(* CoDeSys 2.3.9.50 project: PLC_1111.pro *)
(* Libraries: standard.lib 5.6.98 12:03:02, TcEtherCAT.lib*1.12.15 17:38:26, TcUtilities.lib 3.2.16 16:08:58, TcBase.lib 14.5.09 12:14:08, FB_DateTime.lib 15.2.16 04:06:26, COMlibV2.lib 24.2.14 00:15:46, TcSystem.lib 7.6.16 11:01:22, TcBaseMath.lib 27.7.04 12:07:56, TcMath.lib 23.9.04 15:15:30, TcSystemCX.lib*6.12.13 20:18:08, SysLibVisu.lib 7.7.04 18:17:22, SysLibTargetVisu.lib 16.6.08 16:24:26, TcSUPS.lib 7.6.16 11:50:06 *)

(* Global variable list: Alarms *)
VAR_GLOBAL

	bFeedinfCylFwdRsError:BOOL;
	bErrorRstHmi:BOOL;

	bAGripperConeAllignError: BOOL;
	bAGripCheckDownBuzzer: BOOL;
	sMessage_ServoGripperDown: STRING;

	bQACartonFeedingPistonValve1: BOOL;
	bQACartonFeedingPistonValve2: BOOL;
	bQACartonStopPiston: BOOL;

	bA3COneCrossed: BOOL;
	bA6ConeCrossed: BOOL;
	c18_ConeCounter1: CTU;
	bMCCycleStarted: BOOL;
	bAError: BOOL;
	bAError1: BOOL;
	bSeparatorVerticalPistonEndRsSensed: BOOL;
	bChkEndSensor: BOOL;
	bAConeFeddCylFwdRsError: BOOL;
	bAWrap_1PistRsError: BOOL;
	bAWrap_2PistRsError: BOOL;
	bAWrap_3PistRsError: BOOL;
	bAForwPistRsError: BOOL;
	bASealTopRsError: BOOL;
	bASealTopPistRsError: BOOL;
	bASealSepaX_axisRsError: BOOL;
	bASealSepaY_axisRsError: BOOL;
	bATiltPistRsError: BOOL;
	bAReversPistnRsError: BOOL;
	bAColumnPushPistnRsError: BOOL;
	bAConeEjectPistnRsError: BOOL;
	bASepaHoriForwdFwdEndRsError: BOOL;
	bASepaHoriForwdEndRsError: BOOL;
	bASepaVertiEndPistnRsError: BOOL;
	bASepaHoriRevValveRsError: BOOL;
	bALenghtTightHomeSenRsError: BOOL;
	bABreadthTightHomeSenRsError: BOOL;
	bAGrossWtSenRsError: BOOL;
	bACartonSenRsError: BOOL;
	HmiEmptyCartonPiston: STRING(80);
	bAWrap_PistRsError: BOOL;
	bASealBottomRsError: BOOL;
	SealTopBottomRsError: BOOL;
	SealConeMiss: STRING;
	bConeMissBit: BOOL;
	bAColoumnConeSenError: BOOL;
	bASepVerticalCylRevRsErrChkBit: BOOL;
	bASepaVerCylhomeRsError: BOOL;
	bAL_BTightHomeSenRsError: BOOL;
	GrossWtReedSwBit: BOOL;
	bAGrossWtHomeSenRsError: BOOL;
	bARowStoppHomeSenRsError: BOOL;
	bAPolythinSheetError: BOOL;
	bASepVerticalCylEndRsErrChkBit: BOOL;
	bASupplyPressureError: BOOL;
	baConePtrsentAtWrapConv: BOOL;
	bSealConveyerConePresent: BOOL;
	HmiConeAtSealConveyer: STRING;
	bConeAtMatrixConveter: BOOL;
	bCartonFullDetectbit: BOOL;
	SeparatorAlertbit: BOOL;
	bAFlimNotLoaded: BOOL;
	bFilmErrClear: BOOL;
	bAFirst3ConeAtRowConeCount: BOOL;
	bGrossWieghtNokTemp: BOOL;
	GrossWtAlarm: STRING;
	SealingUnitAlert: BOOL;
	PressureSeparatorAlert: BOOL;
	PistonAlertAlarm: BOOL;
	GripperUnitAlert: BOOL;
	GrossWeightAlert: BOOL;
	ERROR_ALERT: BOOL;
	SealBitAlert: BOOL;
	bAConeMissAtMatricConv: BOOL;
	bHmiColourChangeBit: BOOL;
	bHmiColourChangeBit2: BOOL;
	bAConeAtFullConveyor: BOOL;
	bEmptyCartonDetectError: BOOL;
	HMIEmptyCartonDetectErr: STRING;
	bAEmergencyPressed: BOOL;
	bAConeMissErrorAtWrpConv: BOOL;
	bWrapConvStopped2: BOOL;
	bACheckWrappConvError1: BOOL;
	bACheckWrappConvError2: BOOL;
	bACheckWrappConvError3: BOOL;
	bACheckWrappConvError4: BOOL;
	InterLockCounterRESET: BOOL;
	bCone1LockBit: BOOL;
	bA6conesPushedTemp: BOOL;
	bAConeFeedCylStart: BOOL;
	bWrapConvStopped3: BOOL;
	bAByPassOn2: BOOL;
	bConeMiss3AtWrapConv: BOOL;
	bWrapConvStopped4: BOOL;
	bConeMiss4AtWrapConv: BOOL;
	bAWrapConeCyl123_23: BOOL;
	bCount_ConvLockBit: BOOL;
	bCount_ConvLockBit2: BOOL;
	bCount_ConvLockBitTemp: BOOL;
	FileCreateTemp: BOOL;
	rGrossWeighToReport: REAL;
	bServoOff: BOOL;
	sSupplyPressuremsg: STRING;
	bTLBlinkOn: BOOL;
	PopUp: BOOL;
	bAByPassOn3: BOOL;
	bConeMiss2AtWrapConvtEMP: BOOL;
	CountB_Hmi: INT;
	bA3ConeCrossed_24: BOOL;
	SealBitAlert_24: BOOL;
	bAFilm1Loaded_24_7Cone: BOOL;
	bAFilm1Loaded_24_6Cone: BOOL;
	bAFilm1Loaded_24_5Cone: BOOL;
	bAFilm1Loaded_24_4Cone: BOOL;
	bAFilm1Loaded: BOOL;
	bAFilm2Loaded: BOOL;
	bAFilm3Loaded: BOOL;
	bAFilm1Loaded_24_8Cone: BOOL;
	SealingSafety: BOOL;
	bACheckWrappConvError5: BOOL;
	SensorCheck123: BOOL;
	bAConeMissErrorAtWrpConvTemp1_24: BOOL;
	bAConeMissErrorAtWrpConvTemp2_24: BOOL;
	bAConeMissErrorAtWrpConvTemp3_24: BOOL;
	bAConeMissErrorAtWrpConvTemp4_24: BOOL;
	SensorCheck56: BOOL;
	SensorCheck78: BOOL;
	bWrapConvStopped3_24: BOOL;
	bWrapConvStopped4_24: BOOL;
	bAConeMissErrorAtWrpConvTemp5_24: BOOL;
	bWrapConvStopped4_24exp: BOOL;
	bWrapConvStopped1_24exp: BOOL;
	TON_4_24: TON;
	TON_6_24: TON;
	TON_8_24: TON;
	TON_5_24: TON;
	TON_9_24: TON;
	TON_10_24: TON;
	TON_11_24: TON;
	TON_12_24: TON;
	TON_13_24: TON;
	mybit2: BOOL;
	HmiFullCartonAtConveyer_sensor: STRING;
	bHmiColourChangeBit2_24: BOOL;
	AlarmBitArray: STRING;
	bACheckWrappConv: BOOL;
	var_7: STRING;
	bAinterlockinit: BOOL;
	bAConvStartBit: BOOL;
	test50: BOOL;
	bANo_ErrorBit: BOOL;
END_VAR

(* Global variable list: Common *)
VAR_GLOBAL

	bConeAtWrppingConveyor: BOOL;
	sendOver1:BOOL;
	sendOver2:BOOL;
	sendOver3:BOOL;
	sendOver4:BOOL;
	b2_4SetHmi: BOOL;
	tSealDyl: TIME;
	SealDelay: TON;
	b3ConeSealOver: BOOL;
	bIConeCountSensorVal: INT;
	SealDelay1: TON;
	tSealDyl1: TIME;
	SealDelay2: TON;
	tSealDyl2: TIME;
(*============El6022=================*)

	sSendString : STRING;
	sRecvString : STRING;
	nSendASC:BYTE;
	(* 	I/O variables for a PC-COM port *)

	bAConeUnderWeight: BOOL;
	iACounterA_PV: INT;
	bACounterAReset: BOOL;
	bACounterBReset: BOOL;
	iACounterB_PV: INT;
	iACounterTilt_PV: INT;
	bAresetHmi: BOOL;
	CounterTilt: CTU;
	bAtiltGoHome: BOOL;
	bA5thConeFeedStart: BOOL;
	bAWrappingConvStartAuto: BOOL;
	bAWrappingConvStart: BOOL;
	bAWrappingConvStart1: BOOL;
	bAWrappingConvStart2: BOOL;
	bAWrappingConvStart3: BOOL;
	bAWrappingConvStart4: BOOL;
	bAWrappingConvStart5: BOOL;
	bAWrapConeCyl2: BOOL;
	bA3ConeWrappOver: BOOL;
	bASeal3ConeStart: BOOL;
	bA8thConeWrappOver: BOOL;
	bA6thConeWrappOver: BOOL;
	bA4thWrappOver: BOOL;
	bAutoModeHmi: BOOL;
	bManualModeHmi: BOOL;
	bAColumnPushPistonStart1: BOOL;
	bAColumnPushPistonStart2: BOOL;
	bAMatrixConvStart1: BOOL;
	bAMatrixConvStart2: BOOL;
	bARowStopperMotorRevStart: BOOL;
	bAGripperSeqover: BOOL;
	bAServoDownDone: BOOL;
	bAServoDownDone2: BOOL;

(*

	iarrEcMasterNetId AT %I*: T_AmsNetIdArr;
	nEcMasterSlaveCountCfg AT %I*: UINT;
	bStart: BOOL;
	nTotalSlaves: INT;
	nSalveinfo: ARRAY [0..ISLAVEADDR_ARR_SIZE] OF ST_SlaveStateInfo;
	Iout1 AT%Q*:BOOL;
*)
(*test======*)


	FB_EcGetAllSlaveStates: FB_EcGetAllSlaveStates;
	bEthrcatinfo: BOOL;
	All_slave_Staus_Busy: BOOL;
	All_slave_Staus_Err: BOOL;
	All_slave_Staus_Err_ID: UDINT;
	iNumOfSlavesRead: INT;
	arrSlaveStates: ARRAY [0..10] OF ST_EcSlaveState;

	bAEmptyCartonConvContinue: BOOL;
	bA4thConeFeedStart23: BOOL;
	bA4thConeFeedStartAuto23: BOOL;
	bA6thConeFeedStartAuto23: BOOL;
	bAtiltGoHome3_23: BOOL;

	CounterTilt23: CTU;
	bAtiltGoHome2_23: BOOL;
	bAtiltGoHome1_23: BOOL;
	bAWrappingConvStart1_23: BOOL;
	bAWrappingConvStart4_23: BOOL;
	bAWrappingConvStart3_23: BOOL;
	bAWrappingConvStart2_23: BOOL;
	bA6ConeWrappOver23: BOOL;
	bAColumnPushPistonStart2_23: BOOL;
	bAColumnPushPistonStart1_23: BOOL;

	bAConvFirstStart: BOOL;
	bAServoFwdStart: BOOL;
	bAServoUpAuto: BOOL;
	bAConePickDone: BOOL;
	bAServoDown1Done: BOOL;

	bAPlaceOver: BOOL;
	bAServoFwdStart2: BOOL;
	bAConvSecStart: BOOL;
	bAUnitAWeighOk: BOOL;
	bASeparatorUnitEnable: BOOL;
	bAServoUpDone: BOOL;

	bAFirstSetToMatrix: BOOL;
	bAConvFirstStartUnitB: BOOL;
	bAUnitBWeighOk: BOOL;

	bAConvSecStartUnitB: BOOL;
	bQAFeedingConveyorMotorB: BOOL;
	bQAFeedingConveyorMotorA: BOOL;
	bA3Pushed: BOOL;
	bAconvReayTemp: BOOL;
	bAconvReayTemp2: BOOL;
	bA6conesPushed: BOOL;
	WCPReady: BOOL;
	InterLockCounter: CTU;
	bATiltEnable1: BOOL;

	InterLockCounterStart: BOOL;
	bAWrapConvStarted: BOOL;
	bAInterlockCountStart: BOOL;


	b4thConePushed: BOOL;
	bAconvReayTemp3: BOOL;
	bAconvReadyTemp3: BOOL;
	b6thConePushed_24: BOOL;
	bAconvReadyTemp4: BOOL;
	b8thConesPushed: BOOL;
	bAconvReadyTemp5: BOOL;
	bATiltEnable1_24: BOOL;
	bAConeFeedPistonLockOk: BOOL;

	bATiltEnable2_24: BOOL;
	bAWrapConvReady_24: BOOL;
	bATiltEnable3_24: BOOL;
	bACartonReady_24: BOOL;
	bAResetEnabled: BOOL;
	bRFwdRevPistonRst: BOOL;
	bRTiltPistonReset: BOOL;
	CounterTilt23Rst1: BOOL;
	bACartonReady_23: BOOL;
	bResetRowStopper: BOOL;

	bSealConvIntOver: BOOL;
	bSealConvStart: BOOL;
	bSealConvStart1: BOOL;
	bSealConvStart2: BOOL;
	bASecondSetToMatrix: BOOL;
	bSealConvStart3: BOOL;
	bAConvReady: BOOL;
	bASealConvEnd1: BOOL;
	bASealConvEnd2: BOOL;
	bSaelUnitIntOver: BOOL;
	bWCSStart1: BOOL;
	bWCSStart2: BOOL;
	bWCSStart3: BOOL;
	bMCStart1: BOOL;
	bOneSetReached: BOOL;
	bMCStart2: BOOL;
	bRowStopperAt23Pos: BOOL;
	bATiltPistonInHome: BOOL;
	bSealConvStart1_24: BOOL;
	bSealConvStart2_24: BOOL;
	bSealConvStart3_24: BOOL;
	bASealConvEnd1_24: BOOL;
	bASealConvEnd2_24: BOOL;
	bWCSStart1_24: BOOL;
	bWCSStart2_24: BOOL;
	bRowStopperAt24Pos: BOOL;
	iarrEcMasterNetId: T_AmsNetIdArr ;
	nEcMasterSlaveCountCfg AT %I*: UINT;
	nSalveinfo: ARRAY [0..ISLAVEADDR_ARR_SIZE] OF ST_SlaveStateInfo;

	iRemote2State: INT;
	bRetUnitAStart: BOOL;
	bUnitARowStopperStarted: BOOL;
	bMCStartInAuto: BOOL;
	bStartCartonCov: BOOL;
	bAStartCartonCov: BOOL;

	bRetUnitBStart: BOOL;
	bUnitBRowStopperStarted: BOOL;
	bAOneMinConvStart: BOOL;
	bStartConeFeedConvInBypass: BOOL;
	bUnitBCounterRst: BOOL;
	bASeparatorUnitEnable3: BOOL;
	bASeparatorUnitEnable2: BOOL;
	bASeparatorUnitEnable1: BOOL;
	bQARowStopperMotorRev1: BOOL;
		bAConeOnMatrixConv: BOOL;
	HmiConeOnMatxConvey: STRING;
	bAFilmLoadedCom: BOOL;
	HmiPolyThinFeedErr: STRING;
	bARCartanConvOn: BOOL;
	bOneMinConvOver: BOOL;
	bAWrapConeCyl123: BOOL;
	bAByPassOn: BOOL;
	bA6thConeFeedStart23: BOOL;
	iTotalLayers: INT;
	Count_Hmi: DINT;
	SealingOver: BOOL;
	SealingOver1: BOOL;
	bAFirstConeReached: BOOL;
	Interlockfor_1Cone_24: BOOL;
	Interlockfor_5Cone_24: BOOL;
	Interlockfor_7Cone_24: BOOL;
	UnitACone3Sensing: BOOL;
	UnitACone2Sensing: BOOL;
	UnitACone1Sensing: BOOL;
	UnitACone1_Move: BOOL;
	UnitACone1Sensing_2: BOOL;
	UnitACone2Sensing_2: BOOL;
	UnitACone3Sensing_2: BOOL;
	UnitACone2_Move: BOOL;
	UnitACone3_Move: BOOL;
	UnitA_3_ConeSensed: BOOL;
	R_TRIG_3ConeSensing: R_TRIG;
	iATotalNoOfCones: INT;
	bAUnitBConeCrossing_24: BOOL;
	UnitAConeCrossCount: CTU;
	UnitBCompleteCheckCount_24: CTU;
	Message1_24: STRING;
	sMessage_24: STRING;
	sMessage_23: STRING;
	sMessage_23_Feeding: STRING;
	sMessage_23_Forwad_rev: STRING;
	sMessage_23_Tilting: STRING;
	sMessage_Wrapping: STRING;
	sMessage_Sealing: STRING;
	sMessage_Colomn: STRING;
	sMessage_Gripper: STRING;
	sMessage_Carton: STRING;
	sMessage_Separator: STRING;
	(*FB_S_UPS_CX51x0_1: FB_S_UPS_CX51x0;*)
	bACheckWrappConvError1_23: BOOL;
	bACheckWrappConvError4_23: BOOL;
	bACheckWrappConvError2_23: BOOL;
	bACheckWrappConvError3_23: BOOL;
	mybit1: BOOL;
	temp1: REAL;
	temp2: REAL;
	temp3: REAL;
	temp4: REAL;
	mybit3: BOOL;
	mybit4: BOOL;
	var_1: REAL;
	var_5: REAL;
	bAFeedingConvOff: BOOL;
	bAFeedingConvOff_1: BOOL;
	bQSealBitAlert: BOOL;
	bQSealBitAlert_24: BOOL;
	bA3ConeWrappOver_24: BOOL;
	SealConeMissAlet_24: BOOL;
END_VAR


VAR_GLOBAL CONSTANT
	iSLAVEADDR_ARR_SIZE:DINT:= 256;
END_VAR
(*
VAR_GLOBAL RETAIN
	iTotalLayersHold AT %Q*: INT;
END_VAR *) 
VAR_GLOBAL PERSISTENT
	iTotalLayersHold: INT;
END_VAR

(* Global variable list: Hmi *)
VAR_GLOBAL
	bAllOuputOff: BOOL;
(*	sSettingArray AT %Q*:ARRAY[0..20] OF SETTING; *)
	i:INT;
	sMillNameHmi: STRING(80) := 'INDO TEXNOLOGY';
	AddressLine1Hmi: STRING(80);
	AddressLine2Hmi: STRING(80);
	AddressLine3Hmi: STRING;
	sAddressLine1Hmi: STRING(80) :=' ONDIPUDUR';
	sAddressLine2Hmi: STRING(80) := 'COIMBATORE';
	sAddressLine3Hmi: STRING(80) := 'INDIA';
	bEmptyConeSubOnHmi: BOOL;
	bEmptyConeSubEnabled: BOOL;
	bEmptyConeSubOffHmi: BOOL;
	bAutoRetrivalOnHmi: BOOL;
	bAutoRetrivalEnabled: BOOL;
	bAutoRetrivalOffHmi: BOOL;
	bPrintAutoOnHmi: BOOL;
	bPrintAutoEnabled: BOOL;
	bPrintAutoOffHmi: BOOL;
	PrintDefaultWeightOnHmi: BOOL;
	PrintDefaultWeightOnEnabled: BOOL;
	PrintDefaultWeightOffHmi: BOOL;
	NegToleranceOnHmi: BOOL;
	NegToleranceEnabled: BOOL;
	NegToleranceOffHmi: BOOL;



	Recipe_Var: ARRAY [1..2] OF Recipe;

	DateTimeVar: STRING;
	LogMonth: STRING(80);
	LogYear: STRING(80);
	logDay: STRING(80);
	sStation1ActiveAlarms: STRING(80);
	OperatorName: STRING;

	bEmptyConeSubEnableHMI: BOOL;
	bAEmptyConeSubEnabled: BOOL;
	bEmptyConeSubDisableHMI: BOOL;
	bAutoRetrivalEnableHMI: BOOL;
	bAAutoRetrivalEnabled: BOOL;
	bAutoRetrivalDisableHMI: BOOL;
	bAutoPrintEnableHMI: BOOL;
	bAAutoPrintEnabled: BOOL;
	bAutoPrintDisableHMI: BOOL;
	bDefaultWeighPrintEnableHMI: BOOL;
	bDefaultWeighPrintDisableHMI: BOOL;
	bADefaultWeighPrintEnabled: BOOL;
	bNegToletanceEnableHMI: BOOL;
	bNegToletanceDisableHMI: BOOL;
	bANegToletanceEnabled: BOOL;
	bADayComplete: BOOL;
	bADayStart: BOOL;
	bAutoSealingEnableHMI: BOOL;
	bAAutoSealEnabled: BOOL;
	sCityTownHmi: STRING(80);
	sCountryHmi: STRING(80);
	GrossWeightHmi: REAL;
	NetToleranceHmi: REAL;
	sDescriptionHmi: STRING(80);
(*	SCountHmi: INT;  *)

	iCountHmi: STRING;
	iCartoNoHmi: INT;
	sPackingTypeHmiTemp: STRING(80);
	sMaterialTypeHmiTemp: STRING(80);
	iConeDiaHmi: INT;
	iHieghtHmi: INT;
	iWeightHmi: INT;
	iTipColorHmi: STRING;
	INoOfRowsHmi: INT;
	iNoOfColoumsHmi: INT;
	NoOfLayersHmi: INT;
	iCortonWeightHmi: INT;
	iCartonHmi: INT;
	iLenghtHmi: INT;
	iNoOfConeHmi: INT;
	iNetWeightHmi: REAL;


(*==================*)


	bBlink_Time: BOOL;
	File_Path: STRING;

	bCloseAttachmentList: BOOL;
	bPauseHmi: BOOL;
	bAPauseSeq: BOOL;
	bResumeHmi: BOOL;


	sStringArray:ARRAY [1..cnMaxStrings] OF STRING(300);

	Pgm_NoHmi: INT;
	bNoHmi: BOOL;
	bHidePopUp: BOOL;
	bPauseYesHmi: BOOL;
	bPauseNoHmi: BOOL;

	SealComDlyTemp: TIME;
	wTodayToHmi: STRING;
	bLoadPgm: BOOL;
	bLoadPgmHmi: BOOL;
	bAutoSealingHmi: BOOL;
	bAutoSealOn: BOOL;
	bCartonPackingOn: BOOL;
	bPallettePackingOn: BOOL;
	bCartonPackingHmi: BOOL;
	bPallettePackingHmi: BOOL;
	bConeHmi: BOOL;
	bConeOn: BOOL;
	bCheeseOn: BOOL;
	bCheeseHmi: BOOL;
	bNewRecipeHmi: BOOL;
	Var_PgmNo: INT;
	Var_Description: STRING;

(*==========new variables===========*)
	SaveRecipeHmi: BOOL;
	bCreateNew: BOOL;
	PgmNoDis1: INT;
	PgmNameDis: STRING;
	bModel1Hmi: BOOL;
	PgmNameDis1: STRING(80);
	PgmNameDis2: STRING(80);
	bModel2Hmi: BOOL;
	PgmNoDis3: INT;
	PgmNameDis3: STRING;
	PgmNoDis4: INT;
	PgmNameDis4: STRING;
	PgmNoDis5: INT;
	PgmNoDis6: INT;
	PgmNameDis5: STRING;
	PgmNameDis6: STRING;
	bModel3Hmi: BOOL;
	bModel4Hmi: BOOL;
	bModel5Hmi: BOOL;
	bModel6Hmi: BOOL;
	bEditRecipeHmi: BOOL;
	bEditRecipeEnabled: BOOL;
	bSaveRecipeHmi: BOOL;
	rPickPosMinHmi: REAL := 0.00;
	iDropVeloHmi: REAL;
	PosAct: DINT;
	rServiActPosHmi: REAL;
	b2_3SetHmi: BOOL;
	diVeloActHmi: DINT;
	bStopHmi: BOOL;
	bRetUnitARst: BOOL;
	bGripperOpenHmi: BOOL;
	bGrippercCloseHmi: BOOL;
	sMCStatus: STRING;
	iDropPosHmi: REAL;
	bJogNegHmi: BOOL;
	bJogPositiveHmi: BOOL;
	bJogNegativeHmi: BOOL;
	sRetreivalAStatus: STRING;
	sRetreivalBStatus: STRING;
	bGWPistonOnHmi: BOOL;
	bGWPistonOffHmi: BOOL;
	bRCOnHmi: BOOL;
	bRCOffHmi: BOOL;
	bWeightAckHmi: BOOL;
	bInitializeHmi: BOOL;
	bServoHomeHmi: BOOL;
	rGrossWtTolHmi: REAL;
	bRstHmi: BOOL;
	OpCountHmi: INT;
	bloadRecipeHmi: BOOL;
	rGrossTollHmi: REAL;
	iAPartCountToHmi AT %Q*: INT;
	HmiYAxisPiston: STRING(80);
	HmiXAxisPiston: STRING(80);
	HMISealTopPiston: STRING(80);
	HMISealBotPiston: STRING(80);
	HMIForwdPiston: STRING(80);
	HMIFeedPiston: STRING(80);
	HMIWrapPiston1: STRING(80);
	HMIWrapPiston2: STRING(80);
	HMIWrapPiston3: STRING(80);
	ConeMissAlarm: STRING(80);
	bErrorReset: BOOL;
	HmiTiltPiston: STRING(80);
	HmiReverPiston: STRING(80);
	HmiColuPushrPiston: STRING(80);
	HmiConeEjePiston: STRING(80);
	HmiSepHorizPiston: STRING(80);
	HmiSepVertiPiston: STRING(80);
	HmiSepHoriRevPiston: STRING(80);
	HmiLengthPiston: STRING(80);
	HmiBreadthPiston: STRING(80);
	HmiServoHome: STRING(80);
	HmiGrossWtPiston: STRING(80);
	HmiColoumConeSen: STRING;
	HmiSepVeticCylHomeRsError: STRING;
	HmiGrossWtHomePiston: STRING;
	HmiWrapConvStatus: STRING;
	HmiConeAtMatrixConveyer: STRING;
	HmiFullCartonAtConveyer: STRING;
	bAIntStarted: BOOL;
	HMISeparatorPaperDetec: STRING;
	CounterTilt23_CV_HMI: INT;
	HmiFilmLoadErr: STRING;
	bSheetNotFeeded: STRING;
	bEmergency: BOOL;
	sDATEFinal: STRING;
	sShitToReport: STRING;
	sFinalGrossWt: STRING(80);
	bAIntBlinkAuto: BOOL;
	bALayer1Selected: BOOL;
	bALayer2Selected: BOOL;
	bALayer3Selected: BOOL;
	bMCCycleStartedHold: BOOL;
	RowStopperCountvalue: DINT;



	iLotNoHmi: DWORD;
	bStopEnable: BOOL;
	ITotalSample: DINT;
	iCartonSample: DWORD;
END_VAR
VAR_GLOBAL CONSTANT
	MAX_CSV_ROWS 			: UDINT := 100;
	MAX_CSV_COLUMNS 		: UDINT := 5;
	MAX_CSV_FIELD_LENGTH	: UDINT := 100;

	cnMaxStrings:	INT:=1000;




END_VAR
(*
VAR_GLOBAL RETAIN
	iPickPosHmi AT %Q*: REAL;
	rPickVeloHmi AT %Q*: REAL;
	rDropVeloHmi AT %Q*: REAL;
	iDropPos1Hmi AT %Q*: REAL;
	iDropPos2Hmi AT %Q*: REAL;
	iDropPos3Hmi AT %Q*: REAL;


	bLayer1SelectHmi AT %Q*: BOOL;
	bLayer2SelectHmi AT %Q*: BOOL;
	bLayer3SelectHmi AT %Q*: BOOL;
	iTotalCones AT %Q*: DINT;
END_VAR*)
VAR_GLOBAL PERSISTENT
	iTotalCones: DINT;
	iPickPosHmi: REAL;
	rPickVeloHmi: REAL;
	rDropVeloHmi: REAL;
	iDropPos1Hmi: REAL;
	iDropPos2Hmi: REAL;
	iDropPos3Hmi: REAL;
	bLayer1SelectHmi: BOOL;
	bLayer2SelectHmi: BOOL;
	bLayer3SelectHmi: BOOL;
	sSettingArray: ARRAY [0..20] OF SETTING;
	bAShift1Hour: BOOL;
	bAShift2Hour: BOOL;
	bAShift3Hour: BOOL;
	Shift1MinFrom_HMI: WORD;
	Shift2MinFrom_HMI: WORD;
	Shift3MinFrom_HMI: WORD;
	Shift1MinTo_HMI: WORD;
	Shift2MinTo_HMI: WORD;
	Shift3MinTo_HMI: WORD;
	Sfiht1From_Hmi: WORD;
	Sfiht2From_Hmi: WORD;
	Sfiht3From_Hmi: WORD;
	Sfiht1To_Hmi: WORD;
	Sfiht2To_Hmi: WORD;
	Sfiht3To_Hmi: WORD;
END_VAR

(* Global variable list: Inputs_Gripper *)
VAR_GLOBAL



(******************EL1809(Gripper)*********************)



	bIColumnconeDetection AT %I*: BOOL;
	bIColumnPushPistonHome AT %I*: BOOL;
	bIColumnPushPistonEnd AT %I*: BOOL;
	bIRowConeCountSensor AT %I*: BOOL;
	bIRowConeDetection AT %I*: BOOL;
	bIColumnStopperHome AT %I*: BOOL;
	bIColumnStopper1 AT %I*: BOOL;
	bIColumnStopper2 AT %I*: BOOL;

	bIColumnStopper3 AT %I*: BOOL;
	bIRowStopperHome AT %I*: BOOL;
	bIRowStopper1 AT %I*: BOOL;
	bIRowStopper2 AT %I*: BOOL;
	bIRowStopper3 AT %I*: BOOL;
	bICartonFeedingPistonHome AT %I*: BOOL;
	bICartonFeedingPistonEnd AT %I*: BOOL;
	bIEmptyCartonDetectionSensor AT %I*: BOOL;




(******************EL1809(Gripper)*********************)




	bISeparatorDetectionSensor AT %I*: BOOL;
	bISeparatorPickupDetectionSensor AT %I*: BOOL;
	bICartonPosition1 AT %I*: BOOL;
	bICartonPosition2 AT %I*: BOOL;
	bICartonPosition3 AT %I*: BOOL;
	bISeparatorHorizontalPistonHome AT %I*: BOOL;
	bISeparatorHorizontalPistonEnd AT %I*: BOOL;
	bISeparatorVerticalPistonHome AT %I*: BOOL;


	bISeparatorVerticalPistonEnd AT %I*: BOOL;
	bIGripperVerticalHome AT %I*: BOOL;
	bIGripperVerticalEnd AT %I*: BOOL;
	bILengthTightPistonHome AT %I*: BOOL;
	bIBreadthTightPistonHome AT %I*: BOOL;
	bIConeEjectionPistonHome AT %I*: BOOL;
	bIConeEjectionPistonEnd AT %I*: BOOL;
	bIFullCartonCountingSensor AT %I*: BOOL;


(******************EL1004(Gripper)*********************)

	bIGrossWtDeductSensor AT %I*: BOOL;
	bIGrossWtPistonHome AT %I*: BOOL;
	bIGrossWtPistonEnd AT %I*: BOOL;
	bIGripperConeDetection AT %I*: BOOL;

	iActCounter AT %I*: UDINT;


	b2_3_ACaron: BOOL;
	b2_3_BCarton: BOOL;
	b2_3_ACarton: BOOL;

END_VAR

VAR_GLOBAL PERSISTENT
	b2_3_ACartonHMI: BOOL;
	b2_3_BCartonHMI: BOOL;
END_VAR

(* Global variable list: Inputs_Main *)
VAR_GLOBAL


(******************EL1809(Matrix)*********************)

	bIConeFeedingPistonHome AT %IX0.0: BOOL;
	bIConeFeedingPistonEnd AT %IX0.1: BOOL;
	bIConeOrientationTop AT %IX0.2: BOOL;

	bIForwardPistonHome AT %IX0.3: BOOL;
	bIForwardPistonEnd AT %IX0.4: BOOL;
	bIReversePistonHome AT %IX0.5: BOOL;
	bIReversePistonEnd AT %IX0.6: BOOL;
	bITiltingHome AT %IX0.7: BOOL;
	bITiltingEnd AT %IX1.0: BOOL;
	bIWrappingChannelPiston1_Home AT %IX1.1: BOOL;
	bIWrappingChannelPiston1_End AT %IX1.2: BOOL;
	bIWrappingChannelPiston2_Home AT %IX1.3: BOOL;
	bIWrappingChannelPiston2_End AT %IX1.4: BOOL;
	bIWrappingChannelPiston3_Home AT %IX1.5: BOOL;
	bIWrappingChannelPiston3_End AT %IX1.6: BOOL;
	bISpare AT %IX1.7:BOOL;

(******************EL1809(Matrix)*********************)

	bIWrappingCone1 AT %IX2.0: BOOL;
	bIWrappingCone2 AT %IX2.1: BOOL;
	bIWrappingCone3 AT %IX2.2: BOOL;
	bIWrappingFilmTensionPlate_1 AT %IX2.3: BOOL;
	bIWrappingFilmTensionPlate_2 AT %IX2.4: BOOL;
	bIWrappingFilmTensionPlate_3 AT %IX2.5: BOOL;
	bISealingTopPistonHome AT %IX2.6: BOOL;
	bISealingTopPistonEnd AT %IX2.7: BOOL;
	bISealingBottomPistonHome AT %IX3.0: BOOL;
	bISealingBottomPistonEnd AT %IX3.1: BOOL;
	bIConeCountSensor AT %IX3.2: BOOL;
	bISealingSeparatorYAxisHome AT %IX3.3: BOOL;
	bISealingSeparatorYAxisEnd AT %IX3.4: BOOL;
	bISealingSeparatorXAxisHome AT %IX3.5: BOOL;
	bISealingSeparatorXAxisEnd AT %IX3.6: BOOL;
	bIManualSealing  AT %IX3.7: BOOL;

(******************EL1809(Matrix)*********************)

	bISealingReverseConeSwitch  AT %IX4.0: BOOL;
	bIPressureSwitch   AT %IX4.1: BOOL;
	bIEmergencySwitch   AT %IX4.2: BOOL;
	bIKeySwitch AT %IX4.3: BOOL;
	bIAutoManual AT %IX4.4: BOOL;
	bIMcStart AT %IX4.5: BOOL;
	bIMcStop AT %IX4.6: BOOL;

(**************************End***********************************)



	statusWord AT %I*: UINT;
	bConeMiss1AtWrapConv: BOOL;
	bConeMiss2AtWrapConv: BOOL;
END_VAR

(*
VAR_GLOBAL PERSISTENT
	SealComDly1 AT %Q*: INT;
END_VAR
VAR_GLOBAL RETAIN PERSISTENT
	ghjnk AT %Q*: INT;
END_VAR
*)



VAR_GLOBAL PERSISTENT
	SealComDly1: INT;
	ghjnk: INT;
END_VAR

(* Global variable list: Inputs_RetrivalA_B *)
VAR_GLOBAL

(*******************EL1809(Retrival A & B )*********************)

	bIUnitA_RowStopperHome  AT %IX10.0: BOOL;
	bIUnitA_RowStopperEnd	 AT %IX10.1: BOOL;
	bIUnitB_RowStopperHome	 AT %IX10.2: BOOL;
	bIUnitB_RowStopperEnd	 AT %IX10.3: BOOL;
	bIUnitA_StartPB 		AT %IX10.4: BOOL;
	bIUnitB_StartPB  		AT %IX10.5: BOOL;
	bIUnitB_LiftPistonHome		AT %IX10.6: BOOL;
	bIUnitB_LiftPistonEnd 		AT %IX10.7:BOOL;
	bIUnitAConedetection1 		AT %IX11.0: BOOL;
	bIUnitAConedetection2		 AT %IX11.1: BOOL;
	bIUnitAConedetection3 AT %IX11.2: BOOL;
	bIUnitAConeCrossing AT %IX11.3: BOOL;
	bIUnitBConedetection1  AT %IX11.4: BOOL;
	bIUnitBConedetection2  AT %IX11.5: BOOL;
	bIUnitBConedetection3 AT %IX11.6: BOOL;
	bIUnitBConeCrossing AT %IX11.7:BOOL;

(******************EL1004(Retrival A & B )*********************)

	bIUnitC_LiftPistonHome AT %IX12.0:BOOL;
	bIUnitC_LiftPistonEnd  AT %IX12.1:BOOL;
	bIUnitC_CartonStopForWeight AT %IX12.2:BOOL;
	bISapre14 AT %IX12.3:BOOL;
END_VAR

(* Global variable list: Manual *)
VAR_GLOBAL




		bQMConeFeedingPistonValve :BOOL;
		bQMForwardPistonValve  :BOOL;
		bQMReversePistonValve :BOOL;
		bQMWrappingChannelPistonValve1:BOOL;
		bQMWrappingChannelPistonValve2:BOOL;
		bQMWrappingChannelPistonValve3 :BOOL;
		bQMSealingTopPistonValve :BOOL;
		bQMSealingBottomPistonValve:BOOL;


		bQMFeedingConveyorMotor :BOOL;
		bQMWrappingConveyorMotor :BOOL;
		bQMSealingConveyorMotor :BOOL;
		bQMMatrixConveyorMotor :BOOL;
		bQMFilmRollerMotor1 :BOOL;
		bQMFilmRollerMotor2 :BOOL;
		bQMFilmRollerMotor3 :BOOL;




		bQMRowStopperMotorForward  :BOOL;
		bQMRowStopperMotorReverse:BOOL;
		bQMColumnStopperMotorForward :BOOL;
		bQMColumnStopperMotorReverse:BOOL;
		bQMSealingSeparatorYAxisPistonValve :BOOL;
		bQMSealingSeparatorXAxisPistonValve :BOOL;
		bQMConeTiltingPistonValve :BOOL;
		bQMColumnPushPistonValve:BOOL;

		bQMSeparatorHorizontalPistonValveFwd :BOOL;                     (*X or Y*)
		bQMSeparatorVerticalPistonValve :BOOL;                                   (*X or Y*)
		bQMCartonFeedingPistonValve :BOOL;
		bQMConeEjectionPistonValve :BOOL;
		bQMLengthTightPistonValve :BOOL;
		bQMBreadthTightPistonValve:BOOL;
		bQMEmptyCartonConveyorMotor :BOOL;
		bQMCartonConveyorMotor :BOOL;





		bQMVacuumPistonValve  :BOOL;
		bQMSeparatorHorizontalPistonValveRev  :BOOL;
		bQMSpare1  :BOOL;
		bQMSpare2 :BOOL;


	bQMUnitA_LiftPistonValve:BOOL;
	bQMUnitB_LiftPistonValve: BOOL;
	bQMUnitA_RowStopperMotorForward :BOOL;
	bQMUnitA_RowStopperMotorReverse :BOOL;
	bQMUnitB_RowStopperMotorForward :BOOL;
	bQMUnitB_RowStopperMotorReverse:BOOL;
	bQMUnitC_FullCartonConveyor :BOOL;
	bQMUnitC_LiftPistonValve :BOOL;


	bUA_LiftCylOnHmi: BOOL;
	bUA_LiftCylOffHmi: BOOL;
	bUB_LiftCylOnHmi: BOOL;
	bUB_LiftCylOffHmi: BOOL;
	bUA_RowStopperMotorFwd: BOOL;
	bUA_RowStopperMotorFwdOnHmi: BOOL;
	bUA_RowStopperMotorFwdOffHmi: BOOL;
	bUA_RowStopperMotorRevOnHmi: BOOL;
	bUB_RowStopperMotorFwdOnHmi: BOOL;
	bUB_RowStopperMotorRevOnHmi: BOOL;
	bUC_FullCartonConv: BOOL;
	bUC_FullCartonConvOnHmi: BOOL;
	bUC_FullCartonConvOffHmi: BOOL;
	bUC_LiftCylOnHmi: BOOL;
	bUC_LiftCylOffHmi: BOOL;

	bCFPistonOnHmi: BOOL;
	bCFPistonOffHmi: BOOL;
	bFPValveOnHmi:BOOL;
	bFPValveOffHmi:BOOL;
	bRPValveOnHmi:BOOL;
	bRPValveOffHmi:BOOL;
	bWrappingCPV1OnHmi:BOOL;
	bWrappingCPV1OffHmi:BOOL;
	bWrappingCPV2OnHmi:BOOL;
	bWrappingCPV2OffHmi:BOOL;
	bWrappingCPV3OnHmi:BOOL;
	bWrappingCPV3OffHmi:BOOL;
	bSealingTopPVOnHmi:BOOL;
	bSealingTopPVOffHmi:BOOL;
	bSealingBottomPVOnHmi:BOOL;
	bSealingBottomPVOffHmi:BOOL;
	bFCMotorOnHmi:BOOL;
	bFCMotorOffHmi:BOOL;
	bWCMotorOnHmi:BOOL;
	bWCMotorOffHmi:BOOL;

	bSCMotorOnHmi: BOOL;
	bSCMotorOffHmi: BOOL;
	bMCMotorOnHmi: BOOL;
	bMCMotorOffHmi: BOOL;
	bFRMotor2OnHmi: BOOL;
	bFRMotor2OffHmi: BOOL;
	bFRMotor1OnHmi: BOOL;
	bFRMotor1OffHmi: BOOL;
	bFRMotor3OnHmi: BOOL;
	bFRMotor3OffHmi: BOOL;
	bRSMotorForwardOnHmi: BOOL;
	bRSMotorForwardOffHmi: BOOL;
	bRSMotorRevOnHmi: BOOL;
	bRSMotorRevOffHmi: BOOL;
	bCSMotorFwdOnHmi: BOOL;
	bCSMotorFwdOffHmi: BOOL;
	bCSMotorRevOnHmi: BOOL;
	bCSMotorRevOffHmi: BOOL;
	bSSYAxisPistonValveOnHmi: BOOL;
	bSSYAxisPistonValveOffHmi: BOOL;
	bSSXAxisPistonValveOnHmi: BOOL;
	bSSXAxisPistonValveOffHmi: BOOL;
	bCTPistonValveOnHmi: BOOL;
	bCTPistonValveOffHmi: BOOL;
	bCPushPistonValveOnHmi: BOOL;
	bCPushPistonValveOffHmi: BOOL;
	bSHPistonValveOnHmi: BOOL;
	bSHPistonValveOffHmi: BOOL;
	bSVPistonValveOnHmi: BOOL;
	bSVPistonValveOffHmi: BOOL;
	bCPistonValveOnHmi: BOOL;
	bCPistonValveOffHmi: BOOL;
	bCEPistonValveOnHmi: BOOL;
	bCEPistonValveOffHmi: BOOL;
	bLTPistonValveOnHmi: BOOL;
	bLTPistonValveOffHmi: BOOL;
	bBTightPistonValveOnHmi: BOOL;
	bBTightPistonValveOffHmi: BOOL;
	bECCMotorOnHmi: BOOL;
	bECCMotorOffHmi: BOOL;
	bCCMotorOnHmi: BOOL;
	bCCMotorOffHmi: BOOL;
	bVPValveOnHmi: BOOL;
	bVPValveOffHmi: BOOL;
	bSHPistonValveREVOnHmi: BOOL;
	bSHPistonValveREVOffHmi: BOOL;
	bQMSeparatorHorizontalPistonValveFOR: BOOL;
	bQMColumnPushPistonValveY: BOOL;
	bCPushPistonValveYOnHmi: BOOL;
	bCPushPistonValveYOffHmi: BOOL;
	bMManualSealOn: BOOL;
	bQMLengthPistonValve: BOOL;
	bQMBreathPistonValve: BOOL;
	bQMGrossWtPiston: BOOL;
	bQMRollerConvMotor: BOOL;
	bGWPistonOffHmi1: BOOL;
END_VAR

(* Global variable list: OutpusMain *)
VAR_GLOBAL



		(*===============EL2809 Matrix ===========*)


		bQConeFeedingPistonValve AT %QX0.0 :BOOL;
		bQForwardPistonValve AT %QX0.1 :BOOL;
		bQReversePistonValve AT %QX0.2 :BOOL;
		bQConeTiltingPistonValve AT %QX0.3:BOOL;
		bQWrappingChannelPistonValve1 AT %QX0.4:BOOL;
		bQWrappingChannelPistonValve2 AT %QX0.5:BOOL;
		bQWrappingChannelPistonValve3 AT %QX0.6:BOOL;
		bQSealingTopPistonValve AT %QX0.7:BOOL;

		bQSealingBottomPistonValve  AT %QX1.0:BOOL;
		bQSealingSeparatorYAxisPistonValve AT %QX1.1:BOOL;
		bQSealingSeparatorXAxisPistonValve AT %QX1.2:BOOL;
		bQFeedingConveyorMotor AT %QX1.3:BOOL;
		bQWrappingConveyorMotor AT %QX1.4:BOOL;
		bQFilmRollerMotor1 AT %QX1.5:BOOL;
		bQFilmRollerMotor2 AT %QX1.6:BOOL;
		bQFilmRollerMotor3 AT %QX1.7:BOOL;





		(*===============EL2004 Main ===========*)


		bQSealingConveyorMotorFWD AT %QX2.0 :BOOL;
		bQSealingConveyorMotorREV AT %QX2.1 :BOOL;
		bQTLGreen AT %QX2.2 :BOOL;
		bQTLAmber AT %QX2.3:BOOL;


		(*===============EL2809 Main ===========*)



		bQTLRed AT %QX3.0:BOOL;
		bQBuzzer AT %QX3.1:BOOL;
		bQSpare5 AT %QX3.2:BOOL;
		bQSpare6 AT %QX3.3:BOOL;

(*===============EL2809  Gripper ===========*)



		bQColumnPushPistonValveX AT %Q*:BOOL;
		bQColumnPushPistonValveY AT %Q*:BOOL;
		bQSeparatorHorizontalPistonValveFWD AT %Q*:BOOL;
		bQSeparatorHorizontalPistonValveRev AT %Q*:BOOL;
		bQSeparatorVerticalPistonValve AT %Q*:BOOL;
		bQLengthTightPistonValve AT %Q*:BOOL;
		bQBreadthTightPistonValve  AT %Q*:BOOL;
		bQConeEjectionPistonValve  AT %Q*:BOOL;



		bQCartonFeedingPistonValve  AT %Q*:BOOL;

		bQVacuumPistonValve  AT %Q*:BOOL;
		bQColumnStopperMotorForward AT %Q*:BOOL;
		bQColumnStopperMotorReverse AT %Q*:BOOL;
		bQRowStopperMotorForward AT %Q*:BOOL;
		bQRowStopperMotorReverse AT %Q*:BOOL;
		bQMatrixConveyorMotor AT %Q*:BOOL;
		bQCartonConveyorMotor AT %Q*:BOOL;


	(*===============EL2004 Gripper===========*)

		 bQEmptyCartonConveyorMotor AT %Q*:BOOL;
		 bQGrossWtPiston AT %Q*:BOOL;
		 bQRollerConvMotor AT %Q*:BOOL;
		bQGrossWieghtOkIndi AT %Q*: BOOL;
		bQCartonStopPiston AT %Q*: BOOL;

		iModeControl AT %Q*: UINT;
		iControlWord AT %Q*:UINT;
		diTargetVelocity AT %Q*:DINT;
		diTargetPosition AT %Q*:DINT;






	iControlWord1 AT %Q*: UINT;

	bQSealingConveyorMotorFEV AT %QX2.1: BOOL;
END_VAR
(*
VAR_GLOBAL RETAIN
	vbngh AT %Q*: INT;
	SealComDly AT %Q*: REAL := 2.00;
	testvar AT %Q*: INT;
	bAutoModeOn AT %Q*: BOOL;
	bManualModeOn AT %Q*: BOOL;
END_VAR *)
VAR_GLOBAL PERSISTENT
	bAutoModeOn: BOOL;
	bManualModeOn: BOOL;
	testvar: INT;
	SealComDly: REAL:=2.00;
	vbngh: INT;
	b2_4SetHmiSelected: BOOL;
	b2_3SetHmiSelected: BOOL;
END_VAR

(* Global variable list: OutpusMainFlags *)
VAR_GLOBAL



		(*===============EL2809 Matrix + Gripper===========*)


		bQAConeFeedingPistonValve :BOOL;
		bQAForwardPistonValve  :BOOL;
		bQAReversePistonValve :BOOL;
		bQAWrappingChannelPistonValve1:BOOL;
		bQAWrappingChannelPistonValve2:BOOL;
		bQAWrappingChannelPistonValve3:BOOL;
		bQASealingTopPistonValve :BOOL;
		bQASealingBottomPistonValve:BOOL;

		(*bQAColumnPushPistonValve :BOOL; ======not in use=======*)
		bQAFeedingConveyorMotor :BOOL;
		bQAWrappingConveyorMotor:BOOL;
		bQASealingConveyorMotor :BOOL;
		bQAMatrixConveyorMotor :BOOL;
		bQAFilmRollerMotor1 :BOOL;
		bQAFilmRollerMotor2 :BOOL;
		bQAFilmRollerMotor3 :BOOL;



		(*===============EL2809 Matrix + Gripper===========*)


		bQARowStopperMotorForward  :BOOL;
		bQARowStopperMotorReverse :BOOL;
		bQAColumnStopperMotorForward :BOOL;
		bQAColumnStopperMotorReverse :BOOL;
		bQASealingSeparatorYAxisPistonValve:BOOL;
		bQASealingSeparatorXAxisPistonValve:BOOL;
		bQAConeTiltingPistonValve :BOOL;
		bQAColumnPushPistonValve:BOOL ;
		bQAColumnPushPistonValveY:BOOL;

		bQASeparatorHorizontalPistonValveFwd :BOOL;
		bQASeparatorVerticalPistonValve :BOOL;
		bQACartonFeedingPistonValve :BOOL;
		bQAConeEjectionPistonValve :BOOL;
		bQALengthTightPistonValve :BOOL;
		bQABreadthTightPistonValve:BOOL;
		bQAEmptyCartonConveyorMotor:BOOL;
		bQACartonConveyorMotor :BOOL;



		(*===============EL2004 Matrix + Gripper===========*)


		bQAVacuumPistonValve  :BOOL;
		bQASeparatorHorizontalPistonValveREV  :BOOL;
		bQASpare1  :BOOL;
		bQASpare2 :BOOL;





(*============= EL2008===============*)



	bQAUnitA_LiftPistonValve  :BOOL;
	bQAUnitB_LiftPistonValve : BOOL;
	bQAUnitA_RowStopperMotorForward :BOOL;
	bQAUnitA_RowStopperMotorReverse :BOOL;
	bQAUnitB_RowStopperMotorForward :BOOL;
	bQAUnitB_RowStopperMotorReverse :BOOL;
	bQAUnitC_FullCartonConveyor :BOOL;
	bQAUnitC_LiftPistonValve: BOOL;


	bQAConeTiltingPistonValve1: BOOL;
	bQAConeTiltingPistonValve2: BOOL;
	bQASealingConveyorMotor1: BOOL;
	bQASealingConveyorMotor2: BOOL;
	bQAUnitA_LiftPistonValve1: BOOL;
	bQAUnitA_LiftPistonValve2: BOOL;
	bQAUnitA_RowStopperMotorForward1: BOOL;
	bQAUnitA_RowStopperMotorReverse1: BOOL;
	bQAUnitA_RowStopperMotorForward2: BOOL;
	bQAUnitA_RowStopperMotorReverse2: BOOL;
	bQAUnitB_LiftPistonValve1: BOOL;
	bQAUnitA_RowStopperMotorFwd1: BOOL;
	bQAUnitA_RowStopperMotorRev1: BOOL;
	bQAUnitA_RowStopperMotorFwd2: BOOL;
	bQAUnitB_RowStopperMotorFwd1: BOOL;
	bQAUnitB_RowStopperMotorFwd2: BOOL;
	bQAUnitB_RowStopperMotorRev1: BOOL;
	bQAFeedingConveyor1_23: BOOL;
	bQAFeedingConveyor2_23: BOOL;
	bQAFeedingConveyor3_23: BOOL;
	bQAFeedingConveyor1_24: BOOL;
	bQAFeedingConveyor2_24: BOOL;
	bQAFeedingConveyor3_24: BOOL;
	bQAWrappingConveyorMotor1: BOOL;
	bQAWrappingConveyorMotor2: BOOL;
	bQAWrappingConveyorMotor3: BOOL;
	bQAWrappingConveyorMotor4: BOOL;
	bQAWrappingConveyorMotor5: BOOL;
	bQAWrappingConveyorMotor3_23: BOOL;
	bQAWrappingConveyorMotor4_23: BOOL;
	bQAMatrixConveyor1: BOOL;
	bQAMatrixConveyor2: BOOL;
	sMatrixConvStatus: STRING;

	bQAConeFeedingPistonOnAuto2: BOOL;
	bQAConeFeedingPistonOnAuto1: BOOL;
	bA8thoneReachecdWCS: BOOL;
	bAWrappingCone123OnAuto: BOOL;
	bAWrappingCone123_23OnAuto: BOOL;
	bAWrappingCone23OnAuto: BOOL;
	bAWrappingCone23OnAuto1: BOOL;
	bAWrappingCone3OnAuto: BOOL;
	bQAColumnPushPistonValveY1: BOOL;
	bQAColumnPushPistonValveY2: BOOL;
	bQAGrossWtPiston: BOOL;
	bQARollerConvMotor:BOOL;
	bQAGrossWieghtOkIndi: BOOL;


	bQATLRed: BOOL;
	bQABuzzer: BOOL;
	bQATLAmber: BOOL;
	bQATLGreen: BOOL;

	bQAEmptyCartonConveyorMotor1: BOOL;
END_VAR

(* Global variable list: OutputsRetA_B *)
VAR_GLOBAL

	(*============= EL2008===============*)



	bQUnitA_LiftPistonValve AT %Q* :BOOL;
	bQUnitB_LiftPistonValve AT %Q*: BOOL;
	bQUnitA_RowStopperMotorForward AT %Q*:BOOL;
	bQUnitA_RowStopperMotorReverse AT %Q*:BOOL;
	bQUnitB_RowStopperMotorForward AT %Q*:BOOL;
	bQUnitB_RowStopperMotorReverse AT %Q*:BOOL;
	bQUnitC_FullCartonConveyor AT %Q*:BOOL;
	bQUnitC_LiftPistonValve AT %Q*:BOOL;




END_VAR

(* Global variable list: Reset *)
VAR_GLOBAL
	bARSensorHome: BOOL;
	bARsensorHomeOk: BOOL;
	bQRCartonConveyorMotor: BOOL;
	tEmptyCartonCheckDly: TIME;
	bQRWrappingConveyorMotor: BOOL;
	bQRSealingConveyorMotor: BOOL;
	bQRWrappingChannelPistonValve1: BOOL;
	bQRWrappingChannelPistonValve2: BOOL;
	bQRWrappingChannelPistonValve3: BOOL;
	bQRForwardPistonValve: BOOL;
	bQRReversePistonValve: BOOL;
	bQRSealingTopPistonValve: BOOL;
	bQRSealingSeparatorYAxisPistonValve: BOOL;
	bQRSealingSeparatorXAxisPistonValve: BOOL;
	bQRMatrixConveyorMotor: BOOL;
	bConeAtMatrixConveyor: BOOL;
	sUnitAStatus: STRING;
	sWrapConvStatus: STRING;
	sSealConvStatus: STRING;
	bQRSeparatorHorizontalPistonValveRev: BOOL;
	bARWrappingCone123OnRst: BOOL;
	bColumnPushPistonReset: BOOL;
	bWrpConvIntOver: BOOL;
	bSealingUnitIntOver: BOOL;
	bGripperUnitOver: BOOL;
	bAInitializeSeq: BOOL;
	bMatrixConvIntOver: BOOL;
	bIntRowStopper: BOOL;
	bRowStopperMoveAftrInt: BOOL;
	sCartonConvStatus: STRING;
	bClearConeInt: BOOL;
	bRowStopperEndRSError: BOOL;
	bInterLocCounterRst: BOOL;
	bSealingConvBypass: BOOL;
	bQROneMinConvStart: BOOL;
	bACartonOnGrossWtConv: BOOL;
	sOneMinConMsg: STRING;
	bAOneMinConvReady: BOOL;
	sMianAlarmStatus: STRING;
	bAConeOnSealConvAtInitial: BOOL;
END_VAR

(* Global variable list: serial *)
VAR_GLOBAL

	(*sSendString : STRING;
	sRecvString : STRING;
	nSendASC:BYTE;  *)
	(* 	I/O variables for a PC-COM port *)
	COMin_COMport		AT %I* 	: EL6inData22B ;		(* linked to the port in the TwinCAT System Manager *)
	COMout_COMport		AT %Q*	: EL6outData22B;		(* linked to the port in the TwinCAT System Manager *)
	RxBuffer1: ComBuffer;								(* Receive data buffer; used with all receive function blocks *)
	TxBuffer1: ComBuffer;								(* Transmit data buffer; used with all receive function blocks *)
	RxBuffer2: ComBuffer;
	COMin_2_COMport_2 AT %I*: EL6inData22B;
	COMout_2_COMport_2 AT %Q*: EL6outData22B;
	TxBuffer2: ComBuffer;
	rRetUnitAWeight: REAL;
	rRetUnitBWeight: REAL;
	rRetUnitAWeightNok: BOOL;
	rRetUnitBWeightNok: BOOL;
	bAUnitBConeCrossing_2: BOOL;
	COMin_3_COMport_3 AT %I*: EL6inData22B;
	COMout_3_COMport_3 AT %Q*: EL6outData22B;
	TxBuffer3: ComBuffer;
	RxBuffer3: ComBuffer;
	bReadGWieght: BOOL;
	bGrossWieghtOk: BOOL;
	rGrossWeight: REAL;
	tGrossWtCheckDly: TON;
	bGrossWieghtNok: BOOL;
	bWeightChkAgain: BOOL;
	CyclePass: BOOL;
	bACyclePass: BOOL;

	sTIME: STRING(80);
	bFeedConvStopForUnitB: BOOL;
	bAConeFeedConvStop1: BOOL;
	bFeedConvStopForUnitA: BOOL;
	bAConeFeedConvStop2: BOOL;
	UnitACompleteCheckCount: CTU;
	UnitBCompleteCheckCount: CTU;
	iSerialNo: INT;
	F_TRIG_1: F_TRIG;
	bConvStopForRetB: BOOL;

	R_TRIG_1: R_TRIG;
	bStopConvTemp1: BOOL;
	bStopConvTemp2: BOOL;
	bStopTemp1: BOOL;
	UnitBConeCrossCount: CTU;

	GrossWtVariationTemp: REAL;
	rGrossWtVariation: REAL;
	rGrossWtVariationTemp: REAL;
	rNetWtVariation: REAL;
	rWtVariation: REAL;
	bRowStopperIntOver: BOOL;
	bJogStart: BOOL;
	JogStep: INT;

	CTU_2_UnitA: CTU;
	CTU_2_UnitB: CTU;
	bRowStopperAStart: BOOL;
	bRowStopperBStart: BOOL;
	bUnitARSstart: BOOL;
	bRowStopperStart: BOOL;
	UnitA_18_ConeComDly: TON;
	bAFirst3ConeAtRowConeCountTemp: BOOL;
	bAMainIntStarted: BOOL;
	bEmPopUp: BOOL;
END_VAR


(*
VAR_GLOBAL RETAIN
	iTotalpartCount AT %Q*: DINT;
END_VAR *)
VAR_GLOBAL PERSISTENT
	iTotalpartCount: DINT;
END_VAR

(* Global variable list: Servo *)
VAR_GLOBAL
	ModeWrite: INT;
	ModeAct: BYTE;
	bAModeWrite: BOOL;
	bHomingDone: BOOL;
	diTargetVelocity1: DINT;
	bRServoHome: BOOL;
	bRServoHome1: BOOL;
	bIGripperVerticalEndtemp: BOOL;
	rTargetPosFinal: DINT;
	rDropPosFinal: REAL;
	rDropVeloFinal: REAL;
	rTargetPos: REAL;
	rPickVeloFinal: DINT;

	CountServo: INT;
	bAUnitBConeCrossing_1: BOOL;
	bRowStopperGoHome: BOOL;

	bRowStopperGoRst: BOOL;
	JogModeVar: UINT;
	bJogWrite: BOOL;
	iTorqueAct: INT;
	bServoOnCone: BOOL;
	iTorqueActHmi: REAL;
	bServoReachedUp: BOOL;
	iTorqAvg: INT;
	ReadActCur: INT;
	bServoStartedInAuto: BOOL;
	bServoHome: BOOL;
	bRowStopperGoHome1: BOOL;
	CountServoToSepUnit: INT;
	iACountServoToSepUnit: INT;
END_VAR

(* Global variable list: TwinCAT_Configuration *)
(* Generated automatically by TwinCAT - (read only) *)
VAR_CONFIG
	.nEcMasterSlaveCountCfg AT %IB16 : UINT;
	.iAPartCountToHmi AT %QB4 : INT;
	.bIColumnconeDetection AT %IX96.0 : BOOL;	(*  ~ {LinkedWith:TIID^Device 1 (EtherCAT)^Term 15 (EK1100)^Term 16 (EL1809)^Channel 1^Input} *)
	.bIColumnPushPistonHome AT %IX96.1 : BOOL;	(*  ~ {LinkedWith:TIID^Device 1 (EtherCAT)^Term 15 (EK1100)^Term 16 (EL1809)^Channel 2^Input} *)
	.bIColumnPushPistonEnd AT %IX96.2 : BOOL;	(*  ~ {LinkedWith:TIID^Device 1 (EtherCAT)^Term 15 (EK1100)^Term 16 (EL1809)^Channel 3^Input} *)
	.bIRowConeCountSensor AT %IX96.3 : BOOL;	(*  ~ {LinkedWith:TIID^Device 1 (EtherCAT)^Term 15 (EK1100)^Term 16 (EL1809)^Channel 4^Input} *)
	.bIRowConeDetection AT %IX96.4 : BOOL;	(*  ~ {LinkedWith:TIID^Device 1 (EtherCAT)^Term 15 (EK1100)^Term 16 (EL1809)^Channel 5^Input} *)
	.bIColumnStopperHome AT %IX96.5 : BOOL;	(*  ~ {LinkedWith:TIID^Device 1 (EtherCAT)^Term 15 (EK1100)^Term 16 (EL1809)^Channel 6^Input} *)
	.bIColumnStopper1 AT %IX96.6 : BOOL;	(*  ~ {LinkedWith:TIID^Device 1 (EtherCAT)^Term 15 (EK1100)^Term 16 (EL1809)^Channel 7^Input} *)
	.bIColumnStopper2 AT %IX96.7 : BOOL;	(*  ~ {LinkedWith:TIID^Device 1 (EtherCAT)^Term 15 (EK1100)^Term 16 (EL1809)^Channel 8^Input} *)
	.bIColumnStopper3 AT %IX97.0 : BOOL;	(*  ~ {LinkedWith:TIID^Device 1 (EtherCAT)^Term 15 (EK1100)^Term 16 (EL1809)^Channel 9^Input} *)
	.bIRowStopperHome AT %IX97.1 : BOOL;	(*  ~ {LinkedWith:TIID^Device 1 (EtherCAT)^Term 15 (EK1100)^Term 16 (EL1809)^Channel 10^Input} *)
	.bIRowStopper1 AT %IX97.2 : BOOL;	(*  ~ {LinkedWith:TIID^Device 1 (EtherCAT)^Term 15 (EK1100)^Term 16 (EL1809)^Channel 11^Input} *)
	.bIRowStopper2 AT %IX97.3 : BOOL;	(*  ~ {LinkedWith:TIID^Device 1 (EtherCAT)^Term 15 (EK1100)^Term 16 (EL1809)^Channel 12^Input} *)
	.bIRowStopper3 AT %IX97.4 : BOOL;	(*  ~ {LinkedWith:TIID^Device 1 (EtherCAT)^Term 15 (EK1100)^Term 16 (EL1809)^Channel 13^Input} *)
	.bICartonFeedingPistonHome AT %IX97.5 : BOOL;	(*  ~ {LinkedWith:TIID^Device 1 (EtherCAT)^Term 15 (EK1100)^Term 16 (EL1809)^Channel 14^Input} *)
	.bICartonFeedingPistonEnd AT %IX97.6 : BOOL;	(*  ~ {LinkedWith:TIID^Device 1 (EtherCAT)^Term 15 (EK1100)^Term 16 (EL1809)^Channel 15^Input} *)
	.bIEmptyCartonDetectionSensor AT %IX97.7 : BOOL;	(*  ~ {LinkedWith:TIID^Device 1 (EtherCAT)^Term 15 (EK1100)^Term 16 (EL1809)^Channel 16^Input} *)
	.bISeparatorDetectionSensor AT %IX98.0 : BOOL;	(*  ~ {LinkedWith:TIID^Device 1 (EtherCAT)^Term 15 (EK1100)^Term 17 (EL1809)^Channel 1^Input} *)
	.bISeparatorPickupDetectionSensor AT %IX98.1 : BOOL;	(*  ~ {LinkedWith:TIID^Device 1 (EtherCAT)^Term 15 (EK1100)^Term 17 (EL1809)^Channel 2^Input} *)
	.bICartonPosition1 AT %IX98.2 : BOOL;	(*  ~ {LinkedWith:TIID^Device 1 (EtherCAT)^Term 15 (EK1100)^Term 17 (EL1809)^Channel 3^Input} *)
	.bICartonPosition2 AT %IX98.3 : BOOL;	(*  ~ {LinkedWith:TIID^Device 1 (EtherCAT)^Term 15 (EK1100)^Term 17 (EL1809)^Channel 4^Input} *)
	.bICartonPosition3 AT %IX98.4 : BOOL;	(*  ~ {LinkedWith:TIID^Device 1 (EtherCAT)^Term 15 (EK1100)^Term 17 (EL1809)^Channel 5^Input} *)
	.bISeparatorHorizontalPistonHome AT %IX98.5 : BOOL;	(*  ~ {LinkedWith:TIID^Device 1 (EtherCAT)^Term 15 (EK1100)^Term 17 (EL1809)^Channel 6^Input} *)
	.bISeparatorHorizontalPistonEnd AT %IX98.6 : BOOL;	(*  ~ {LinkedWith:TIID^Device 1 (EtherCAT)^Term 15 (EK1100)^Term 17 (EL1809)^Channel 7^Input} *)
	.bISeparatorVerticalPistonHome AT %IX98.7 : BOOL;	(*  ~ {LinkedWith:TIID^Device 1 (EtherCAT)^Term 15 (EK1100)^Term 17 (EL1809)^Channel 8^Input} *)
	.bISeparatorVerticalPistonEnd AT %IX99.0 : BOOL;	(*  ~ {LinkedWith:TIID^Device 1 (EtherCAT)^Term 15 (EK1100)^Term 17 (EL1809)^Channel 9^Input} *)
	.bIGripperVerticalHome AT %IX99.1 : BOOL;	(*  ~ {LinkedWith:TIID^Device 1 (EtherCAT)^Term 15 (EK1100)^Term 17 (EL1809)^Channel 10^Input} *)
	.bIGripperVerticalEnd AT %IX99.2 : BOOL;	(*  ~ {LinkedWith:TIID^Device 1 (EtherCAT)^Term 15 (EK1100)^Term 17 (EL1809)^Channel 11^Input} *)
	.bILengthTightPistonHome AT %IX99.3 : BOOL;	(*  ~ {LinkedWith:TIID^Device 1 (EtherCAT)^Term 15 (EK1100)^Term 17 (EL1809)^Channel 12^Input} *)
	.bIBreadthTightPistonHome AT %IX99.4 : BOOL;	(*  ~ {LinkedWith:TIID^Device 1 (EtherCAT)^Term 15 (EK1100)^Term 17 (EL1809)^Channel 13^Input} *)
	.bIConeEjectionPistonHome AT %IX99.5 : BOOL;	(*  ~ {LinkedWith:TIID^Device 1 (EtherCAT)^Term 15 (EK1100)^Term 17 (EL1809)^Channel 14^Input} *)
	.bIConeEjectionPistonEnd AT %IX99.6 : BOOL;	(*  ~ {LinkedWith:TIID^Device 1 (EtherCAT)^Term 15 (EK1100)^Term 17 (EL1809)^Channel 15^Input} *)
	.bIFullCartonCountingSensor AT %IX99.7 : BOOL;	(*  ~ {LinkedWith:TIID^Device 1 (EtherCAT)^Term 15 (EK1100)^Term 17 (EL1809)^Channel 16^Input} *)
	.bIGrossWtDeductSensor AT %IX100.0 : BOOL;	(*  ~ {LinkedWith:TIID^Device 1 (EtherCAT)^Term 15 (EK1100)^Term 18 (EL1004)^Channel 1^Input} *)
	.bIGrossWtPistonHome AT %IX100.1 : BOOL;	(*  ~ {LinkedWith:TIID^Device 1 (EtherCAT)^Term 15 (EK1100)^Term 18 (EL1004)^Channel 2^Input} *)
	.bIGrossWtPistonEnd AT %IX100.2 : BOOL;	(*  ~ {LinkedWith:TIID^Device 1 (EtherCAT)^Term 15 (EK1100)^Term 18 (EL1004)^Channel 3^Input} *)
	.bIGripperConeDetection AT %IX104.0 : BOOL;
	.iActCounter AT %IB18 : UDINT;
	.statusWord AT %IB22 : UINT;	(*  ~ {LinkedWith:TIID^Device 2 (EL6751)^Box 1 (LXM32AD18N4     )^TxPDO 1^Inputs^Statusword} *)
	.bQColumnPushPistonValveX AT %QX92.0 : BOOL;	(*  ~ {LinkedWith:TIID^Device 1 (EtherCAT)^Term 15 (EK1100)^Term 19 (EL2809)^Channel 1^Output} *)
	.bQColumnPushPistonValveY AT %QX92.1 : BOOL;	(*  ~ {LinkedWith:TIID^Device 1 (EtherCAT)^Term 15 (EK1100)^Term 19 (EL2809)^Channel 2^Output} *)
	.bQSeparatorHorizontalPistonValveFWD AT %QX92.2 : BOOL;	(*  ~ {LinkedWith:TIID^Device 1 (EtherCAT)^Term 15 (EK1100)^Term 19 (EL2809)^Channel 3^Output} *)
	.bQSeparatorHorizontalPistonValveRev AT %QX92.3 : BOOL;	(*  ~ {LinkedWith:TIID^Device 1 (EtherCAT)^Term 15 (EK1100)^Term 19 (EL2809)^Channel 4^Output} *)
	.bQSeparatorVerticalPistonValve AT %QX92.4 : BOOL;	(*  ~ {LinkedWith:TIID^Device 1 (EtherCAT)^Term 15 (EK1100)^Term 19 (EL2809)^Channel 5^Output} *)
	.bQLengthTightPistonValve AT %QX92.5 : BOOL;	(*  ~ {LinkedWith:TIID^Device 1 (EtherCAT)^Term 15 (EK1100)^Term 19 (EL2809)^Channel 6^Output} *)
	.bQBreadthTightPistonValve AT %QX92.6 : BOOL;	(*  ~ {LinkedWith:TIID^Device 1 (EtherCAT)^Term 15 (EK1100)^Term 19 (EL2809)^Channel 7^Output} *)
	.bQConeEjectionPistonValve AT %QX92.7 : BOOL;	(*  ~ {LinkedWith:TIID^Device 1 (EtherCAT)^Term 15 (EK1100)^Term 19 (EL2809)^Channel 8^Output} *)
	.bQCartonFeedingPistonValve AT %QX93.0 : BOOL;	(*  ~ {LinkedWith:TIID^Device 1 (EtherCAT)^Term 15 (EK1100)^Term 19 (EL2809)^Channel 9^Output} *)
	.bQVacuumPistonValve AT %QX93.1 : BOOL;	(*  ~ {LinkedWith:TIID^Device 1 (EtherCAT)^Term 15 (EK1100)^Term 19 (EL2809)^Channel 10^Output} *)
	.bQColumnStopperMotorForward AT %QX93.2 : BOOL;	(*  ~ {LinkedWith:TIID^Device 1 (EtherCAT)^Term 15 (EK1100)^Term 19 (EL2809)^Channel 11^Output} *)
	.bQColumnStopperMotorReverse AT %QX93.3 : BOOL;	(*  ~ {LinkedWith:TIID^Device 1 (EtherCAT)^Term 15 (EK1100)^Term 19 (EL2809)^Channel 12^Output} *)
	.bQRowStopperMotorForward AT %QX93.4 : BOOL;	(*  ~ {LinkedWith:TIID^Device 1 (EtherCAT)^Term 15 (EK1100)^Term 19 (EL2809)^Channel 13^Output} *)
	.bQRowStopperMotorReverse AT %QX93.5 : BOOL;	(*  ~ {LinkedWith:TIID^Device 1 (EtherCAT)^Term 15 (EK1100)^Term 19 (EL2809)^Channel 14^Output} *)
	.bQMatrixConveyorMotor AT %QX93.6 : BOOL;	(*  ~ {LinkedWith:TIID^Device 1 (EtherCAT)^Term 15 (EK1100)^Term 19 (EL2809)^Channel 15^Output} *)
	.bQCartonConveyorMotor AT %QX93.7 : BOOL;	(*  ~ {LinkedWith:TIID^Device 1 (EtherCAT)^Term 15 (EK1100)^Term 19 (EL2809)^Channel 16^Output} *)
	.bQEmptyCartonConveyorMotor AT %QX94.0 : BOOL;	(*  ~ {LinkedWith:TIID^Device 1 (EtherCAT)^Term 15 (EK1100)^Term 20 (EL2004)^Channel 1^Output} *)
	.bQGrossWtPiston AT %QX94.1 : BOOL;	(*  ~ {LinkedWith:TIID^Device 1 (EtherCAT)^Term 15 (EK1100)^Term 20 (EL2004)^Channel 2^Output} *)
	.bQRollerConvMotor AT %QX94.2 : BOOL;	(*  ~ {LinkedWith:TIID^Device 1 (EtherCAT)^Term 15 (EK1100)^Term 20 (EL2004)^Channel 3^Output} *)
	.bQGrossWieghtOkIndi AT %QX94.3 : BOOL;
	.bQCartonStopPiston AT %QX96.0 : BOOL;
	.iModeControl AT %QB6 : UINT;
	.iControlWord AT %QB8 : UINT;
	.diTargetVelocity AT %QB10 : DINT;	(*  ~ {LinkedWith:TIID^Device 2 (EL6751)^Box 1 (LXM32AD18N4     )^RxPDO 3^Outputs^Target velocity} *)
	.diTargetPosition AT %QB14 : DINT;	(*  ~ {LinkedWith:TIID^Device 2 (EL6751)^Box 1 (LXM32AD18N4     )^RxPDO 2^Outputs^Target position} *)
	.iControlWord1 AT %QB18 : UINT;	(*  ~ {LinkedWith:TIID^Device 2 (EL6751)^Box 1 (LXM32AD18N4     )^RxPDO 1^Outputs^Controlword;
													TIID^Device 2 (EL6751)^Box 1 (LXM32AD18N4     )^RxPDO 2^Outputs^Controlword;
													TIID^Device 2 (EL6751)^Box 1 (LXM32AD18N4     )^RxPDO 3^Outputs^Controlword} *)
	.bQUnitA_LiftPistonValve AT %QX94.4 : BOOL;	(*  ~ {LinkedWith:TIID^Device 1 (EtherCAT)^Term 12 (EK1100)^Term 14 (EL2008)^Channel 1^Output} *)
	.bQUnitB_LiftPistonValve AT %QX94.5 : BOOL;	(*  ~ {LinkedWith:TIID^Device 1 (EtherCAT)^Term 12 (EK1100)^Term 14 (EL2008)^Channel 2^Output} *)
	.bQUnitA_RowStopperMotorForward AT %QX94.6 : BOOL;	(*  ~ {LinkedWith:TIID^Device 1 (EtherCAT)^Term 12 (EK1100)^Term 14 (EL2008)^Channel 3^Output} *)
	.bQUnitA_RowStopperMotorReverse AT %QX94.7 : BOOL;	(*  ~ {LinkedWith:TIID^Device 1 (EtherCAT)^Term 12 (EK1100)^Term 14 (EL2008)^Channel 4^Output} *)
	.bQUnitB_RowStopperMotorForward AT %QX95.0 : BOOL;	(*  ~ {LinkedWith:TIID^Device 1 (EtherCAT)^Term 12 (EK1100)^Term 14 (EL2008)^Channel 5^Output} *)
	.bQUnitB_RowStopperMotorReverse AT %QX95.1 : BOOL;	(*  ~ {LinkedWith:TIID^Device 1 (EtherCAT)^Term 12 (EK1100)^Term 14 (EL2008)^Channel 6^Output} *)
	.bQUnitC_FullCartonConveyor AT %QX95.2 : BOOL;	(*  ~ {LinkedWith:TIID^Device 1 (EtherCAT)^Term 12 (EK1100)^Term 14 (EL2008)^Channel 7^Output} *)
	.bQUnitC_LiftPistonValve AT %QX95.3 : BOOL;	(*  ~ {LinkedWith:TIID^Device 1 (EtherCAT)^Term 12 (EK1100)^Term 14 (EL2008)^Channel 8^Output} *)
	.COMin_COMport AT %IB24 : EL6inData22B;
	.COMout_COMport AT %QB20 : EL6outData22B;
	.COMin_2_COMport_2 AT %IB48 : EL6inData22B;
	.COMout_2_COMport_2 AT %QB44 : EL6outData22B;
	.COMin_3_COMport_3 AT %IB72 : EL6inData22B;
	.COMout_3_COMport_3 AT %QB68 : EL6outData22B;
END_VAR

(* Data type in EtherCAT Diag *)
TYPE E_EcCommState : (
	eEcState_UNDEFINED 		:= 0,
	eEcState_INIT 				:= 1,
	eEcState_PREOP 			:= 2,
	eEcState_BOOT 				:= 3,
	eEcState_SAFEOP 			:= 4,
	eEcState_OP 				:= 8
);
END_TYPE

(* Data type *)
TYPE ErrorAlarm_Data :
STRUCT

	Error_No						:STRING;
	SDateF						:STRING;
	sShift						:STRING;
	Time_No					:STRING;

(*	ActualNetWt					:STRING;
	LotNo						:STRING;
	sCount						:STRING;
	StandardGrossWt				:STRING;
	NetWt						:STRING;
	sTolerance					:STRING;
	sEmpConeWt					:STRING; *)

END_STRUCT
END_TYPE

(* Data type *)
TYPE Production_Data :
STRUCT

	S_No						:STRING;
	CartonNo					:STRING;
	SDateF						:STRING;
	sShift						:STRING;
	ActualNetWt					:STRING;
	LotNo						:STRING;
	sCount						:STRING;
	StandardGrossWt				:STRING;
	NetWt						:STRING;
	sTolerance					:STRING;
	sEmpConeWt					:STRING;

END_STRUCT
END_TYPE

(* Data type *)
TYPE Recipe :
STRUCT

	Pgm_No:STRING;
	Description:STRING;
	Count:STRING;
	Lot_No:STRING;
	Carton_No:STRING;
	PackingType:STRING(80);
	MaterialType:STRING(80);
	Cone_Dia:STRING;
	Hight:STRING;
	Weight:STRING;
	TipColor:STRING;
	NoOfRows:STRING;
	NoOfColums:STRING;
	NoOfLayer:STRING;
	CartonW:STRING;
	CartonH:STRING;
	lenght:STRING;
	NoOfCone:STRING;
	NetWeight:STRING;
	GrossWeight:STRING;
	NetTolerance:STRING;

END_STRUCT
END_TYPE

(* Data type *)
TYPE SETTING :
STRUCT
	iPgmNo:INT;
	sDescription:STRING;
	iCount:STRING;
	iLotNo:DWORD;
	iCartonNo:INT;
	bAutoSealing:BOOL;
	bCartonPacking:BOOL;
	bPallettePack:BOOL;
	bCone:BOOL;
	bCheese:BOOL;
	iConeDia:INT;
	iConeHight:INT;
	iConeWeight:INT;
	iTipColor:STRING;
	iNoOfRows:INT;
	iNoOfColoumns:INT;
	iNoOfLayers:INT;
	iCartonwidth:INT;
	iCartonHight:INT;
	iCartonLength:INT;
	iNoOfCones:INT;
	iGrosswt:REAL;
	iNetWt:REAL;
	iNetTol:REAL;
	iGrossTol:REAL;



END_STRUCT
END_TYPE

(* Data type *)
TYPE ST_CSV_Record :
STRUCT
	sName 	: T_MaxString 	:= '';
	nNumber	: UDINT 		:= 0;
	fPos		: LREAL 		:= 0.0;
	bOP		: BOOL 		:= FALSE;
	sDesc		: STRING(40)	:= '';
	data		: ARRAY[0..7] OF STRING;
END_STRUCT
END_TYPE

(* Data type in EtherCAT Diag *)
TYPE ST_SlaveState :
STRUCT
	(* slave state *)
	eEcState 			: E_EcCommState;
	nReserved			: UINT;
	bError				: BOOL;
	bInvalidVPRS		: BOOL;
	nReserved2			: UINT;

	(* link state *)
	bNoCommToSlave	: BOOL;
	bLinkError			: BOOL;
	bMissingLink			: BOOL;
	bUnexpectedLink		: BOOL;
	bPortA				: BOOL;
	bPortB				: BOOL;
	bPortC				: BOOL;
	bPortD				: BOOL;
END_STRUCT
END_TYPE

(* Data type in EtherCAT Diag *)
TYPE ST_SlaveStateInfo :
STRUCT
(*	nIndex 			: DINT;*)
(*	sName 			: STRING; *)		(* name of slave given in System Manager *)
(*	sType 			: STRING;	*)	(* type of slave, e.g. EK1100*)
(*	nECAddr 		: UINT;		*)	(* EtherCAT Slave Addr *)
	bDiagData		: BOOL;			(* DiagData in Slave State *)
(*


ortCRCErrors	: ST_EcCrcErrorEx;*)(* Slave CRC-Errors, separate for each Port *)
(*	nSumCRCErrors	: UDINT;	*)	(* Slave CRC-Errors, sum of all Ports *)
	stState 		: ST_SlaveState;(* EtherCAT State and Link state*)
END_STRUCT
END_TYPE

(* POU MAIN, ST *)
PROGRAM MAIN
VAR
	step: INT;
	testOut: DINT;
	Scale_1: Scale;
	va1: INT;
	va2: INT;
	invar2: DINT;
	invar1: DINT;
	var1: DINT;
	var2: DINT;
	out1: INT;
	out2: INT;
	mainout: INT;

	GetAllSlaveStates: FB_EcGetAllSlaveStates;
	EcGetSlaveState: FB_EcGetSlaveState;
	test: BOOL;
	nTotalSlaves: INT;
	EtherCatInfo_1: EtherCatInfo;

	test1: BYTE;
	test2: BYTE;
	EverRunTimer: TON;
	bIAutoManualTemp: BOOL;
	bManualmode: BOOL;
	JogTimer1: TON;
	bMCReady: BOOL;
	BlinkTimer1: TON;
	BlinkTimer2: TON;


	(*FB_S_UPS_CX51xx_1: FB_S_UPS_CX51x0;*)
	FB_S_UPS_1: FB_S_UPS;
END_VAR
	IF bIMcStart AND bAutoModeOn AND NOT  bServoOff  THEN bMCStartInAuto:=TRUE; bStopEnable:=FALSE;  END_IF

	IF NOT bIEmergencySwitch OR  bIMcStop OR bStopHmi  OR bServoOff  THEN bMCStartInAuto:=FALSE; END_IF


						(*============== Auto/Manual Mode Selection Logic========================*)

		IF bIAutoManual THEN
			bAutoModeOn:=TRUE; bManualModeOn:=FALSE;
		ELSIF  bManualmode  THEN
			bManualModeOn:=TRUE; bAutoModeOn:=FALSE;
		END_IF

		IF bManualModeOn THEN sMCStatus:='Machine in Manual Mode';
		ELSIF bAutoModeOn THEN sMCStatus:='Machine in Auto Mode';
		END_IF

	IF bMCStartInAuto  AND NOT  bIAutoManual THEN bHidePopUp:=TRUE; END_IF

	IF NOT  bMCStartInAuto  AND NOT  bIAutoManual THEN bManualmode:=TRUE; ELSE bManualmode:=FALSE;  END_IF

	IF bHidePopUp AND bPauseYesHmi THEN bManualmode:=TRUE; bHidePopUp:=FALSE; END_IF

	IF bHidePopUp AND bPauseNoHmi THEN  bHidePopUp:=FALSE; END_IF




                                                                                    (*====================Logic for Model Selection===============*)

		IF bAutoModeOn AND b2_4SetHmi THEN
		b2_4SetHmiSelected:=TRUE; b2_3SetHmiSelected:=FALSE;b2_3SetHmi:=FALSE;
		ELSIF bAutoModeOn AND   b2_3SetHmi THEN
		b2_4SetHmiSelected:=FALSE; b2_3SetHmiSelected:=TRUE; b2_4SetHmi:=FALSE;
		END_IF

		IF b2_4SetHmiSelected THEN Message1_24:=' 24  Cones '; END_IF

		IF b2_3SetHmiSelected THEN Message1_24:=' 18  Cones  '; END_IF

		WeightCalc();
		Outputs();
		FlimRollerUnit();
		HMI();
		RowStopperMotor();
		ColumStopperMotor();
		GripperUnitRst();
		Serial();


IF bAutoModeOn THEN

		Servo_Auto();


		PickAndPlaceUnit();
	(*	AlarmSave(); *)
		DataLog_1();
		DataLog_Alarm();
		ColomnPushPiston_XY();
		Matrix_Conveyor();
		CartonConveyor();
		EmptyConveyor();
		SeparatorUnit();
		UnitA_RowStopper24();
		UnitB_RowStopper24();



		OneMinConv();
		Sealing_Unit();
		ConeAllignAlarm();
		Cylinder_Alarm();
		ServoError();
		SeparatorAlarm();

END_IF



	Manual();
	Jogging();

	SDOREAD();
	ServoHoming();
	ServoSetting();


	INT_All();


IF NOT bSealingConvBypass THEN
	Sealing_Conveyor_23();

END_IF


IF b2_3SetHmiSelected THEN
	ConeFeedPiston_23();
	Tilt_Piston_23();
	FwdRevPiston_2_3();
	ConeFeedConvNew_23();
	Wrapping_Unit();
(*
ConeFeedConvNew();*)
END_IF



IF b2_4SetHmiSelected THEN
	Tilt_Piston_24();
	FwdRevPiston_2_4();
	ConeFeedPiston_24();
	ConeFeedConvNew_23();
	UnitA_RowStopper24();
	UnitB_RowStopper24();
	Wrapping_Unit_24();
	Sealing_Conveyor_24();
END_IF




bQAConeTiltingPistonValve:= ( bQAConeTiltingPistonValve2 OR bQAConeTiltingPistonValve1 );

bQASealingConveyorMotor:= ( bQASealingConveyorMotor1 OR bQASealingConveyorMotor2);

bQAUnitA_LiftPistonValve:= ( bQAUnitA_LiftPistonValve1 );

bQAUnitA_RowStopperMotorForward:= ( bQAUnitA_RowStopperMotorForward1 );

bQAUnitA_RowStopperMotorReverse:= ( bQAUnitA_RowStopperMotorReverse1);

bQAFeedingConveyorMotor:= ( bQAFeedingConveyorMotorA OR bQAFeedingConveyorMotorB );

bQAConeFeedingPistonValve:=( bQAConeFeedingPistonOnAuto1 OR bQAConeFeedingPistonOnAuto2 );



                                                                          (*===============ETHERCAT SLAVE STATUS============*)

EtherCatInfo_1(
	arrEcMasterNetId:=iarrEcMasterNetId ,
	bExecute:=TRUE ,
	nSlaveCountCfg:=nEcMasterSlaveCountCfg ,
	iNumOfSlavesRead=>nTotalSlaves ,
	arrSlaveInfo=>nSalveinfo );


                                                    (*============= Remote station 2 EtherCat slave states============================*)
iRemote2State:=EtherCatInfo_1.arrSlaveStates[13].deviceState;

                                                           (*=============Company Logo Popup Window appear logic=============*)
PopUp:=TRUE;

EverRunTimer(IN:=PopUp , PT:=t#2s , Q=> , ET=> );


                                                                          (*=============== JOg Mode Change Logic===========*)

IF bManualModeOn THEN
JogTimer1(IN:=bManualModeOn , PT:=t#100ms , Q=> , ET=> );
IF JogTimer1.Q THEN bJogStart :=TRUE; JogTimer1(IN:=FALSE); END_IF
END_IF

IF bAutoModeOn THEN   bJogStart :=FALSE; JogStep:=0;  END_IF

                                                                                     (*============Tower Lamp Logic============*)


IF bRowStopperIntOver AND bACartonReady_23   AND bMCStartInAuto AND NOT bAError  THEN bMCReady:=TRUE; bMCCycleStarted:=FALSE; END_IF

IF bMCStartInAuto AND bRetUnitAStart OR bRetUnitBStart AND NOT bAError THEN bMCCycleStarted:=TRUE; bMCCycleStartedHold:=TRUE;  bMCReady:=FALSE;  END_IF

IF NOT  bIEmergencySwitch OR bStopHmi OR bIMcStop THEN bMCCycleStartedHold:=FALSE; END_IF


IF bMCStartInAuto   AND  bMCCycleStarted AND bAError1 THEN bAError:=TRUE; ELSE bAError:=FALSE; END_IF


                                                                            (*===============Tower Lamp Logic=======================*)

IF  bMCStartInAuto  AND NOT  bAPauseSeq AND NOT ERROR_ALERT AND NOT bAMainIntStarted   THEN bQATLGreen :=TRUE; bQATLRed:=FALSE;
ELSIF  bStopEnable OR bAEmergencyPressed OR  bServoOff AND NOT   bMCStartInAuto  AND NOT  bAPauseSeq   AND NOT ERROR_ALERT
AND NOT bAMainIntStarted THEN bQATLRed:=TRUE; bQATLGreen:=FALSE;
 END_IF


IF  bStopHmi OR bIMcStop THEN bStopEnable:=TRUE; END_IF



IF bAMainIntStarted  AND NOT bServoOff THEN bTLBlinkOn:=TRUE; bQATLGreen:=FALSE;  ELSE  bTLBlinkOn:=FALSE; END_IF
BlinkTimer1(IN:=(bTLBlinkOn AND NOT BlinkTimer2.Q) , PT:= t#0.5s, Q=> , ET=> );
BlinkTimer2(IN:= BlinkTimer1.Q, PT:=t#1.3s , Q=> , ET=> );

IF BlinkTimer1.Q AND NOT bServoOff THEN bAIntBlinkAuto:=TRUE; ELSE  bAIntBlinkAuto:=FALSE; END_IF

                                                                         (*=============== Servo Power Off Finding Logic===================*)

IF NOT statusWord.4 THEN
bServoOff:=TRUE;
ELSE
bServoOff:=FALSE;
END_IF


FB_S_UPS_1(
	sNetID:= '5.17.63.202.1.1',
	iPLCPort:=801 ,
	iUPSPort:=16#4A8 ,
	tTimeout:= T#5s,
	eUpsMode:= eSUPS_WrPersistData_Shutdown ,
	ePersistentMode:= SPDM_2PASS ,
	tRecoverTime:=T#10s ,
	bPowerFailDetect=> ,
	eState=> );
(*

FB_S_UPS_CX51xx_1(
	sNetID:= ,
	iPLCPort:=AMSPORT_R0_PLC_RTS1 ,
	iUPSPort:= 16#588 ,
	tTimeout:=DEFAULT_ADS_TIMEOUT ,
	eUpsMode:=eSUPS_WrPersistData_Shutdown ,
	ePersistentMode:= FB_S_UPS_CX51xx_1.ePersistentMode ,
	tRecoverTime:= T#10s ,
	bPowerFailDetect=> ,
	eState=> );
*)
END_PROGRAM

(* POU FunctionBlocks/Scale, ST *)
FUNCTION_BLOCK Scale
VAR_INPUT
	INPUT: REAL;
	INPUTMIN: REAL;
	INPUTMAX: REAL;
	OUTPUTMIN: REAL;
	OUTPUTMAX: REAL;
END_VAR

VAR_OUTPUT
	OUTPUT:REAL;
END_VAR

VAR
	INPUT_REAL:REAL;
	INPUTMIN_REAL:REAL;
	INPUTMAX_REAL:REAL;
	OUTPUTMIN_REAL:REAL;
	OUTPUTMAX_REAL:REAL;
	OUTPUT_REAL: REAL;
	TEMP_REAL:REAL;
END_VAR
	INPUT_REAL :=  INPUT;
	INPUTMIN_REAL :=INPUTMIN;
	INPUTMAX_REAL := INPUTMAX;
	OUTPUTMIN_REAL :=OUTPUTMIN;
	OUTPUTMAX_REAL :=OUTPUTMAX;

	IF INPUTMAX_REAL<>INPUTMIN_REAL THEN
		TEMP_REAL		:=	(INPUT_REAL - INPUTMIN_REAL)/(INPUTMAX_REAL - INPUTMIN_REAL);
		OUTPUT_REAL	:=	(TEMP_REAL * (OUTPUTMAX_REAL - OUTPUTMIN_REAL) + OUTPUTMIN_REAL);
	END_IF

	OUTPUT := REAL_TO_INT(OUTPUT_REAL);
END_FUNCTION_BLOCK

(* POU FunctionBlocks/EtherCatInfo, ST *)
FUNCTION_BLOCK EtherCatInfo
VAR_INPUT
		(*NetId*)
		arrEcMasterNetId	: T_AmsNetIdArr;
		bExecute: BOOL;
		nSlaveCountCfg: UINT;
END_VAR
VAR_OUTPUT
		iNumOfSlavesRead: INT;
		arrSlaveInfo 				: ARRAY [0..iSLAVEADDR_ARR_SIZE] OF ST_SlaveStateInfo;
END_VAR
VAR
(*Generate NetId*)
	sEcMasterNetId: T_AmsNetId;
(* Slave States*)
		fbEcGetAllSlaveAddr: FB_EcGetAllSlaveAddr;
	arrSlaveStates: ARRAY [0..ISLAVEADDR_ARR_SIZE] OF ST_EcSlaveState;
	(*Get Slave Adddress*)
		FB_EcGetSlaveState_Terminal:FB_EcGetSlaveState ;
(* -- Get Slave States *)
	fbGetAllSlaveStates			: FB_EcGetAllSlaveStates;
	I: DINT;
	iDiagIndex					: ARRAY [0..3] OF UINT;

END_VAR
(*Generate NetId*)
sEcMasterNetId := F_CreateAmsNetId(nIds := arrEcMasterNetId);

(*Get Slave States*)
fbGetAllSlaveStates(
	sNetId		:='5.42.152.186.2.1'(* sEcMasterNetId*),
	pStateBuf	:= ADR(arrSlaveStates),
	cbBufLen	:= SIZEOF(arrSlaveStates),
	bExecute	:= bExecute,
	tTimeout	:= DEFAULT_ADS_TIMEOUT,
	nSlaves		=> iNumOfSlavesRead
);


	IF NOT fbGetAllSlaveStates.bBusy THEN
		fbGetAllSlaveStates(bExecute:= FALSE);

		IF NOT fbGetAllSlaveStates.bError THEN
			IF iNumOfSlavesRead = nSlaveCountCfg THEN
				FOR I := 0 TO 3 DO
					iDiagIndex[I] := 0;
				END_FOR

		(* split slave state and link state *)
			FOR I := 0 TO MIN(iNumOfSlavesRead, iSLAVEADDR_ARR_SIZE) DO
				(* slave state*)
				arrSlaveInfo[I].stState.eEcState 			:= arrSlaveStates[I].deviceState AND 16#0F;
				arrSlaveInfo[I].stState.bError 			:= arrSlaveStates[I].deviceState.4;
				arrSlaveInfo[I].stState.bInvalidVPRS 		:= arrSlaveStates[I].deviceState.5;
				(* link state *)
				arrSlaveInfo[I].stState.bNoCommToSlave 	:= arrSlaveStates[I].linkState.0;
				arrSlaveInfo[I].stState.bLinkError 			:= arrSlaveStates[I].linkState.1;
				arrSlaveInfo[I].stState.bMissingLink 		:= arrSlaveStates[I].linkState.2;
				arrSlaveInfo[I].stState.bUnexpectedLink	 := arrSlaveStates[I].linkState.3;
				arrSlaveInfo[I].stState.bPortA 			:= arrSlaveStates[I].linkState.4;
				arrSlaveInfo[I].stState.bPortB 			:= arrSlaveStates[I].linkState.5;
				arrSlaveInfo[I].stState.bPortC 			:= arrSlaveStates[I].linkState.6;
				arrSlaveInfo[I].stState.bPortD 			:= arrSlaveStates[I].linkState.7;
				(* DiagData *)
				arrSlaveInfo[I].bDiagData	:= ((arrSlaveStates[I].deviceState AND 16#F0) <> 0) OR
					(((arrSlaveStates[I].deviceState AND 16#0F) > 0) AND ((arrSlaveStates[I].deviceState AND 16#0F) < 8)) OR
					(arrSlaveStates[I].linkState <> 0);

				IF arrSlaveInfo[I].bDiagData THEN
					IF (I=0) THEN
						iDiagIndex[0] := 0;
					ELSE
						IF (iDiagIndex[0] = 0) AND NOT arrSlaveInfo[0].bDiagData THEN
							iDiagIndex[0] :=  DINT_TO_UINT(I);
						END_IF
					END_IF
				END_IF
			END_FOR
		END_IF
	END_IF
	END_IF
END_FUNCTION_BLOCK

(* POU WeightCalc, ST *)
PROGRAM WeightCalc
VAR
	CounterA: CTU;
	R_TRIG_1: R_TRIG;
	CounterB: CTU;
	R_TRIG_2: R_TRIG;
	R_TRIG_3: R_TRIG;

	ConeCountEnable: BOOL;
	InterLockCounterStartTimer: TON;
	TON_3: TON;
	tResetTiner: TON;
	WCPReadyTemp1: BOOL;
	WCPReadyTemp2: BOOL;
	Det: WORD;
	BreadTemp: BOOL;
	ADSREAD_1: ADSREAD;
	SwithOnButtton: BOOL;
	axis1: BOOL;
	RstStep: INT;
	bStopTiltUnit: BOOL;
	rRetUnitTolMax: REAL;
	rRetUnitTolMin: REAL;
	rRetUnitAWeightok: BOOL;

	TON_4: TON;
	rRetUnitAWeightempt: REAL;
	rRetUnitAWeighttemp: REAL;
	TON_5: TON;
	rRetUnitBWeightok: BOOL;
	TON_6: TON;
	TON_7: TON;
	rGrossWtTolMax: REAL;
	rGrossWtTolMin: REAL;
	TON_8: TON;
	bGrossWieghtOkTemp: BOOL;

	Timer1: TON;
	Timer2: TON;
	bMonitor: BOOL;
	bStartBlinker: BOOL;
	UnitAWeightBit: BOOL;
	UnitBWeightBit: BOOL;
	weightCheck: INT;
	Weight1Move: BOOL;
	var_2: REAL;
	Weight3Move: BOOL;
	Timer_3: TON;

	var_3: REAL;
	weightCheck1: INT;
	Weight2Move: BOOL;
	var_4: REAL;
	Weight4Move: BOOL;
	Timer_4: TON;
END_VAR
(*===========Reterival unit weight ok and not ok Logic UNIT-A=================*)

(*==== Weight Max & Min Tolerance Setting==========*)

rRetUnitTolMax:= (sSettingArray[i].iNetWt + sSettingArray[i].iNetTol);

	IF NegToleranceEnabled AND bAutoModeOn THEN
	rRetUnitTolMin:= (sSettingArray[i].iNetWt - sSettingArray[i].iNetTol);
	ELSIF NOT NegToleranceEnabled THEN rRetUnitTolMin:= (sSettingArray[i].iNetWt);
	END_IF
IF rRetUnitAWeight  <= rRetUnitTolMax AND rRetUnitAWeight >=rRetUnitTolMin THEN
rRetUnitAWeightok:=TRUE;
ELSE
rRetUnitAWeightok:=FALSE;
END_IF

IF TON_5.Q   THEN bQAUnitA_LiftPistonValve:=TRUE; END_IF
(*
ELSIF Timer1.Q THEN bQAUnitA_LiftPistonValve:=TRUE; ELSE  bQAUnitA_LiftPistonValve:=TRUE; END_IF
IF  bUnitARowStopperStarted  THEN bStartBlinker:=TRUE; ELSE   bStartBlinker:=FALSE;


Timer1(IN:=(bStartBlinker AND NOT Timer2.Q)  , PT:=t#50ms , Q=> , ET=> );

Timer2(IN:=Timer1.Q , PT:=t#50ms , Q=> , ET=> );
*)
(*=========== Unit A Start after wieght ok logic=================*)

IF bIUnitA_StartPB  AND bQAUnitA_LiftPistonValve AND bAutoModeOn AND NOT bStartConeFeedConvInBypass THEN  bRetUnitAStart:=TRUE; END_IF


(*============Weight stabilization time======================*)


IF rRetUnitAWeightok THEN TON_4(IN:=TRUE , PT:=t#2s , Q=> , ET=> ); ELSE  TON_4(IN:=FALSE); END_IF

(*============== WEIGHT NOT OK DEFINE TIME ( TON_5)=================*)

IF TON_4.Q THEN TON_5(IN:=TRUE , PT:=t#0.5s , Q=> , ET=> ); ELSE TON_5(IN:=FALSE); END_IF

IF bAutoModeOn AND bIUnitA_RowStopperHome AND NOT rRetUnitAWeightok THEN rRetUnitAWeightNok:=TRUE; ELSE rRetUnitAWeightNok:=FALSE;   END_IF
(*
  IF rRetUnitAWeightNok THEN bRetUnitAStart:=FALSE; END_IF
*)


(*===============weight not ok Indicator on logic====================*)

IF rRetUnitAWeightNok THEN bQAUnitB_LiftPistonValve:=TRUE; ELSE  bQAUnitB_LiftPistonValve:=FALSE;  END_IF


(*================ Weight ok feedback to Auto Logic=============*)

IF  rRetUnitAWeightok THEN bAUnitAWeighOk:=TRUE;  ELSE bAUnitAWeighOk:=FALSE; END_IF


(*===========Reterival unit weight ok and not ok Logic UNIT-B =================*)


IF rRetUnitBWeight  <= rRetUnitTolMax AND rRetUnitBWeight >=rRetUnitTolMin THEN
rRetUnitBWeightok:=TRUE;
ELSE
rRetUnitBWeightok:=FALSE;
END_IF

IF TON_7.Q THEN bQAUnitC_FullCartonConveyor:=TRUE; ELSE  bQAUnitC_FullCartonConveyor:=FALSE;  END_IF




(*=========== Unit A Start after wieght ok logic=================*)

IF bIUnitB_StartPB  AND bQAUnitC_FullCartonConveyor AND bAutoModeOn  AND NOT bStartConeFeedConvInBypass
 THEN  bRetUnitBStart:=TRUE; END_IF


(*============Weight stabilization time======================*)


IF rRetUnitBWeightok THEN TON_6(IN:=TRUE , PT:=t#2s , Q=> , ET=> ); ELSE  TON_6(IN:=FALSE); END_IF

(*============== WEIGHT NOT OK DEFINE TIME ( TON_5)=================*)

IF TON_6.Q THEN TON_7(IN:=TRUE , PT:=t#0.5s , Q=> , ET=> ); ELSE TON_7(IN:=FALSE); END_IF

IF bAutoModeOn AND bIUnitB_RowStopperHome AND NOT rRetUnitBWeightok THEN rRetUnitBWeightNok:=TRUE; ELSE rRetUnitBWeightNok:=FALSE;   END_IF
(*
  IF rRetUnitBWeightNok THEN bRetUnitBStart:=FALSE; END_IF
*)


(*===============weight not ok Indicator on logic====================*)


IF rRetUnitBWeightNok THEN bQAUnitC_LiftPistonValve:=TRUE; ELSE  bQAUnitC_LiftPistonValve:=FALSE;  END_IF


(*================ Weight ok feedback to Auto Logic=============*)

IF  rRetUnitBWeightok THEN bAUnitBWeighOk:=TRUE; ELSE bAUnitBWeighOk:=FALSE;  END_IF




(*============================================================================================================================================================*)



(*===================UnitA Cone Count Logic================*)

CounterA(
	CU:=bIUnitAConeCrossing ,
	RESET:=R_TRIG_1.Q ,
	PV:=iACounterA_PV ,
	Q=> ,
	CV=> );

R_TRIG_1(CLK:= bACounterAReset , Q=> );

(*===================UnitB Cone Count Logic================*)

CounterB(
	CU:=bIUnitBConeCrossing ,
	RESET:=R_TRIG_2.Q ,
	PV:=iACounterB_PV ,
	Q=> ,
	CV=> );

R_TRIG_2(CLK:= bACounterBReset , Q=> );






		IF b2_3SetHmiSelected THEN
		iACounterA_PV:=18;
		iACounterB_PV:=18;
		iACounterTilt_PV:=6;

		ELSIF  b2_4SetHmiSelected THEN
		iACounterA_PV:=24;
		iACounterB_PV:=24;
		iACounterTilt_PV:=8;
		END_IF


(*===================UnitA Cone Count Reset Logic================*)



		IF  (*bIUnitA_LiftPistonEnd  AND *) bIUnitA_RowStopperHome AND NOT bIUnitAConeCrossing THEN
		bACounterAReset:=TRUE;
		ELSE
		bACounterAReset:=FALSE;
		END_IF




(*===================UnitB Cone Count Reset Logic================*)



		IF bIUnitB_LiftPistonEnd AND bIUnitB_RowStopperHome AND NOT bIUnitBConeCrossing THEN
		bACounterBReset:=TRUE;
		ELSE
		bACounterBReset:=FALSE;
		END_IF



IF bIWrappingCone1 AND bIWrappingChannelPiston1_Home AND bIWrappingChannelPiston1_Home AND bIWrappingChannelPiston1_Home THEN
ConeCountEnable:=TRUE;
ELSE
ConeCountEnable:=FALSE;
END_IF

(*

InterLockCounterStartTimer(IN:= InterLockCounterStart , PT:=T#0.5s , Q=> , ET=> );
*)

TON_3(IN:=bAInterlockCountStart , PT:= T#0.2s , Q=> , ET=> );

R_TRIG_3(CLK:=TON_3.Q , Q=> );

InterLockCounter(
	CU:=R_TRIG_3.Q ,
	RESET:=InterLockCounterRESET ,
	PV:=6 ,
	Q=> ,
	CV=> );
IF bInitializeHmi  OR bInterLocCounterRst THEN
InterLockCounterRESET:=TRUE;
ELSE
InterLockCounterRESET:=FALSE;
END_IF



IF InterLockCounter.CV=3 AND bA3Pushed THEN
bAconvReayTemp:=TRUE;
END_IF

IF   InterLockCounter.CV=4 AND b4thConePushed AND b2_4SetHmiSelected THEN
bAconvReadyTemp3:=TRUE;
END_IF


IF InterLockCounter.CV=6 AND bA6conesPushed AND b2_3SetHmiSelected THEN
bAconvReayTemp2:=TRUE;
END_IF

IF InterLockCounter.CV = 6 AND b6thConePushed_24 AND  b2_4SetHmiSelected THEN
bAconvReadyTemp4:=TRUE;
END_IF

IF bAconvReayTemp2 THEN
bA6conesPushed:=FALSE;
InterLockCounterRESET:=TRUE;
END_IF


IF  InterLockCounter.CV = 8 AND   bA8thoneReachecdWCS AND b2_4SetHmiSelected THEN
bAconvReadyTemp5:=TRUE;

END_IF

IF bAconvReadyTemp5 THEN
InterLockCounterRESET:=TRUE;
b8thConesPushed:=FALSE;
END_IF


IF   InterLockCounter.CV=0 THEN WCPReady:=TRUE; ELSE   WCPReady:=FALSE; END_IF



IF  NOT  bIEmergencySwitch  OR  bStopHmi OR bIMcStop OR bServoOff  THEN bStopTiltUnit:=TRUE; END_IF

CASE RstStep OF
	0:	IF bStopTiltUnit THEN
		RstStep:=RstStep+1;
		END_IF
	1:	IF bITiltingEnd OR bITiltingHome THEN
		bRFwdRevPistonRst:=TRUE;
		bStopTiltUnit:=FALSE;
		RstStep:=RstStep+1;
		END_IF
	2:	IF bIForwardPistonHome AND bIReversePistonHome THEN
		bRFwdRevPistonRst:=FALSE;
		RstStep:=RstStep+1;
		END_IF
	3:	bRTiltPistonReset:=TRUE;
		RstStep:=RstStep+1;

	4:	IF bITiltingHome THEN
		bRTiltPistonReset:=FALSE;
		RstStep:=0;
		END_IF
END_CASE




SealComDly1;

IF bRetUnitAStart AND NOT bRetUnitBStart  AND NOT UnitBWeightBit THEN UnitAWeightBit:=TRUE; var_1:=rRetUnitAWeight; END_IF
IF bRetUnitBStart AND NOT bRetUnitAStart AND NOT UnitAWeightBit  THEN UnitBWeightBit:=TRUE; var_2:=rRetUnitBWeight; END_IF

CASE  weightCheck OF


	0:	IF  UnitAWeightBit AND NOT UnitBWeightBit THEN
		Weight1Move:=TRUE;
		weightCheck:=1;END_IF

	1:	IF  Weight1Move AND NOT Weight3Move THEN
		var_3:=var_1;
		Weight3Move:=TRUE;
		Weight1Move:=FALSE;

		weightCheck:=2;END_IF

	2:	IF  bACyclePass AND Weight3Move THEN
		 var_5:=var_3;
		weightCheck:=3;END_IF

	3: 	IF Weight3Move THEN Timer_3(IN:=TRUE , PT:= T#1s , Q=> , ET=> );
		IF Timer_3.Q THEN Weight3Move:=FALSE; UnitAWeightBit:=FALSE;Timer_3(IN:=FALSE);
		weightCheck:=0;END_IF END_IF

END_CASE

CASE  weightCheck1 OF

	0:	IF  UnitBWeightBit AND NOT UnitAWeightBit THEN
		Weight2Move:=TRUE;
		weightCheck1:=1;END_IF

	1:	IF  Weight2Move AND NOT Weight4Move THEN
		var_4:=var_2;
		Weight4Move:=TRUE;
		Weight2Move:=FALSE;

		weightCheck1:=2;END_IF

	2:	IF  bACyclePass AND Weight4Move  THEN
		var_5:=var_4;
		weightCheck1:=3;END_IF

	3: 	IF Weight4Move THEN Timer_4(IN:=TRUE , PT:= T#1s , Q=> , ET=> );
		IF Timer_4.Q THEN Weight4Move:=FALSE;UnitBWeightBit:=FALSE; Timer_4(IN:=FALSE);
		weightCheck1:=0;END_IF END_IF

END_CASE

IF NOT bIEmergencySwitch OR bIMcStop OR bServoOff OR   bStopHmi THEN
Weight1Move:=FALSE;
Weight2Move:=FALSE;
Weight3Move:=FALSE;
Weight4Move:=FALSE;
Timer_3(IN:=FALSE);
Timer_4(IN:=FALSE);
UnitAWeightBit:=FALSE;
UnitBWeightBit:=FALSE;
END_IF


ghjnk;
END_PROGRAM

(* POU Outputs, ST *)
	PROGRAM Outputs
VAR
	bQATLAmbertemp: BOOL;
END_VAR
		(*===============EL2809 Main ===========*)


		bQConeFeedingPistonValve   :=   (bQMConeFeedingPistonValve OR bQAConeFeedingPistonValve) ;
		bQForwardPistonValve  :=   (bQMForwardPistonValve OR bQAForwardPistonValve OR bQRForwardPistonValve ) ;
		bQReversePistonValve  :=  bQMReversePistonValve OR bQAReversePistonValve OR bQRReversePistonValve ;
		bQConeTiltingPistonValve :=  ( bQMConeTiltingPistonValve OR bQAConeTiltingPistonValve);
		bQWrappingChannelPistonValve1  :=  bQMWrappingChannelPistonValve1 OR  bQAWrappingChannelPistonValve1 OR bQRWrappingChannelPistonValve1;
		bQWrappingChannelPistonValve2  :=  bQMWrappingChannelPistonValve2 OR bQAWrappingChannelPistonValve2 OR bQRWrappingChannelPistonValve2;
		bQWrappingChannelPistonValve3  :=  bQMWrappingChannelPistonValve3 OR bQAWrappingChannelPistonValve3 OR bQRWrappingChannelPistonValve3;
		bQSealingTopPistonValve  :=  bQMSealingTopPistonValve OR bQASealingTopPistonValve OR bQRSealingTopPistonValve ;




		bQSealingBottomPistonValve  :=  bQMSealingBottomPistonValve OR bQASealingBottomPistonValve  ;
		bQSealingSeparatorYAxisPistonValve:=  (bQMSealingSeparatorYAxisPistonValve OR bQASealingSeparatorYAxisPistonValve OR bQRSealingSeparatorYAxisPistonValve );
		bQSealingSeparatorXAxisPistonValve:=  ( bQMSealingSeparatorXAxisPistonValve OR bQASealingSeparatorXAxisPistonValve OR bQRSealingSeparatorXAxisPistonValve );
		bQFeedingConveyorMotor:=bQMFeedingConveyorMotor OR bQAFeedingConveyorMotor  ;
		bQWrappingConveyorMotor:=bQMWrappingConveyorMotor OR bQAWrappingConveyorMotor OR bQRWrappingConveyorMotor;
		bQFilmRollerMotor1:=bQMFilmRollerMotor1 OR bQAFilmRollerMotor1;
		bQFilmRollerMotor2 :=bQMFilmRollerMotor2 OR bQAFilmRollerMotor2;
		bQFilmRollerMotor3 :=bQMFilmRollerMotor3 OR bQAFilmRollerMotor3;



	(*===============EL2004 Main===========*)


		bQSealingConveyorMotorFWD :=bQMSealingConveyorMotor OR bQASealingConveyorMotor OR bQRSealingConveyorMotor;
		bQSealingConveyorMotorFEV;



	(*==============EL2809   main=========*)

		bQTLRed:=  bQATLRed OR bAIntBlinkAuto;
		bQBuzzer:= bQABuzzer;
		bQTLGreen :=bQATLGreen OR bAIntBlinkAuto ;
		bQTLAmber:=bQATLAmber OR bAIntBlinkAuto ;

;



(*===============EL2809 Gripper===========*)


		bQMatrixConveyorMotor :=bQMMatrixConveyorMotor OR bQAMatrixConveyorMotor OR bQRMatrixConveyorMotor;



		bQRowStopperMotorForward :=bQMRowStopperMotorForward OR bQARowStopperMotorForward ;
		bQRowStopperMotorReverse:=bQMRowStopperMotorReverse OR bQARowStopperMotorReverse;
		bQColumnStopperMotorForward:=bQMColumnStopperMotorForward OR bQAColumnStopperMotorForward   ;
		bQColumnStopperMotorReverse:= ( bQMColumnStopperMotorReverse OR bQAColumnStopperMotorReverse ) ;

		bQColumnPushPistonValveX:=  (bQMColumnPushPistonValve OR bQAColumnPushPistonValve );
		bQColumnPushPistonValveY:=(bQMColumnPushPistonValveY OR bQAColumnPushPistonValveY OR bColumnPushPistonReset);



		bQSeparatorHorizontalPistonValveFwd := ( bQMSeparatorHorizontalPistonValveFwd OR bQASeparatorHorizontalPistonValveFwd) ;                     (*X or Y*)
		bQSeparatorVerticalPistonValve :=  (bQMSeparatorVerticalPistonValve OR bQASeparatorVerticalPistonValve );                                   (*X or Y*)
		bQCartonFeedingPistonValve := (bQMCartonFeedingPistonValve OR bQACartonFeedingPistonValve);
		bQConeEjectionPistonValve:=  (bQMConeEjectionPistonValve  OR bQAConeEjectionPistonValve);
		bQLengthTightPistonValve:=  (bQMLengthTightPistonValve OR bQALengthTightPistonValve );
		bQBreadthTightPistonValve:=  ( bQMBreadthTightPistonValve OR bQABreadthTightPistonValve );
		bQEmptyCartonConveyorMotor:=  ( bQMEmptyCartonConveyorMotor OR bQAEmptyCartonConveyorMotor );
		bQCartonConveyorMotor:=  ( bQMCartonConveyorMotor  OR bQACartonConveyorMotor );

(*============= EL2004===============*)


		bQGrossWtPiston:=(bQAGrossWtPiston OR bQMGrossWtPiston);
		bQRollerConvMotor:=(bQARollerConvMotor OR  bQMRollerConvMotor OR bQROneMinConvStart ) ;

	(*===============EL2004 Matrix + Gripper===========*)


		bQVacuumPistonValve:=  (bQMVacuumPistonValve OR bQAVacuumPistonValve);
		bQSeparatorHorizontalPistonValveRev:=  (bQMSeparatorHorizontalPistonValveRev OR bQASeparatorHorizontalPistonValveRev OR bQRSeparatorHorizontalPistonValveREV ) ;



(*============= EL2008===============*)



	bQUnitA_LiftPistonValve:=  bQAUnitA_LiftPistonValve;
	bQUnitB_LiftPistonValve:=	bQAUnitB_LiftPistonValve  ;
	bQUnitA_RowStopperMotorForward:=bQMUnitA_RowStopperMotorForward OR bQAUnitA_RowStopperMotorForward;
	bQUnitA_RowStopperMotorReverse:= bQMUnitA_RowStopperMotorReverse OR bQAUnitA_RowStopperMotorReverse  ;
	bQUnitB_RowStopperMotorForward:= bQMUnitB_RowStopperMotorForward OR bQAUnitB_RowStopperMotorForward;
	bQUnitB_RowStopperMotorReverse:= bQMUnitB_RowStopperMotorReverse OR bQAUnitB_RowStopperMotorReverse;
	bQUnitC_FullCartonConveyor:= bQMUnitC_FullCartonConveyor OR bQAUnitC_FullCartonConveyor;
	bQUnitC_LiftPistonValve:= bQMUnitC_LiftPistonValve OR bQAUnitC_LiftPistonValve;


bQCartonStopPiston:=bQACartonStopPiston;
END_PROGRAM

(* POU Auto/FlimRollerUnit, ST *)
PROGRAM FlimRollerUnit
VAR
	step: INT;
	bQAFilmRollerMotor1OnAuto: BOOL;
	bQAFilmRollerMotor2OnAuto: BOOL;
	bQAFilmRollerMotor3OnAuto: BOOL;
	F_TRIG_1: F_TRIG;
	F_TRIG_2: F_TRIG;
	F_TRIG_3: F_TRIG;


END_VAR
bQAFilmRollerMotor1:= ( bQAFilmRollerMotor1OnAuto );

bQAFilmRollerMotor2:= ( bQAFilmRollerMotor2OnAuto );

bQAFilmRollerMotor3:=( bQAFilmRollerMotor3OnAuto );


		IF NOT 	bIWrappingFilmTensionPlate_1 AND iRemote2State = 8 THEN
		bQAFilmRollerMotor1OnAuto:=TRUE;
		ELSE
		bQAFilmRollerMotor1OnAuto:=FALSE;
		END_IF


		IF NOT	bIWrappingFilmTensionPlate_2  AND iRemote2State = 8 THEN
		bQAFilmRollerMotor2OnAuto:=TRUE;
		ELSE
		bQAFilmRollerMotor2OnAuto:=FALSE;
		END_IF



		IF NOT	bIWrappingFilmTensionPlate_3   AND iRemote2State = 8 THEN
		bQAFilmRollerMotor3OnAuto:=TRUE;
		ELSE
		bQAFilmRollerMotor3OnAuto:=FALSE;
		END_IF



F_TRIG_1(CLK:=bIWrappingFilmTensionPlate_1 , Q=> );
F_TRIG_2(CLK:=bIWrappingFilmTensionPlate_2 , Q=> );
F_TRIG_3(CLK:=bIWrappingFilmTensionPlate_3 , Q=> );


					(*###################### 1,2,3th Cone Film Loaded in 2*3   ###################*)

IF (bAWrappingCone123OnAuto OR bAWrappingCone123_23OnAuto) AND bAutoModeOn AND b2_3SetHmiSelected  AND F_TRIG_1.Q AND NOT  bIWrappingChannelPiston1_End THEN
bAFilm1Loaded:=TRUE; END_IF
IF( bAWrappingCone123OnAuto OR bAWrappingCone123_23OnAuto) AND bAutoModeOn  AND b2_3SetHmiSelected AND F_TRIG_2.Q AND NOT  bIWrappingChannelPiston2_End THEN
bAFilm2Loaded:=TRUE; END_IF
IF( bAWrappingCone123OnAuto  OR bAWrappingCone123_23OnAuto ) AND bAutoModeOn AND b2_3SetHmiSelected  AND F_TRIG_3.Q AND NOT  bIWrappingChannelPiston3_End THEN
 bAFilm3Loaded:=TRUE; END_IF
IF bAFilm1Loaded AND bAFilm2Loaded AND bAFilm3Loaded AND b2_3SetHmiSelected  THEN
 bAFilmLoadedCom:=TRUE; bAFilm1Loaded:=FALSE; bAFilm2Loaded:=FALSE;bAFilm3Loaded:=FALSE;   END_IF


					(*###################### 1,2,3th Cone Film Loaded in 2*4     ###################*)

IF (bAWrappingCone123OnAuto OR bAWrappingCone123_23OnAuto) AND bAutoModeOn AND b2_4SetHmiSelected  AND F_TRIG_1.Q AND NOT  bIWrappingChannelPiston1_End THEN
bAFilm1Loaded:=TRUE; END_IF
IF( bAWrappingCone123OnAuto OR bAWrappingCone123_23OnAuto) AND bAutoModeOn AND b2_4SetHmiSelected AND F_TRIG_2.Q AND NOT  bIWrappingChannelPiston2_End THEN
bAFilm2Loaded:=TRUE; END_IF
IF( bAWrappingCone123OnAuto  OR bAWrappingCone123_23OnAuto ) AND bAutoModeOn  AND b2_4SetHmiSelected AND F_TRIG_3.Q AND NOT  bIWrappingChannelPiston3_End THEN
 bAFilm3Loaded:=TRUE; END_IF
IF bAFilm1Loaded AND bAFilm2Loaded AND bAFilm3Loaded AND b2_4SetHmiSelected THEN
 bAFilmLoadedCom:=TRUE; bAFilm1Loaded:=FALSE; bAFilm2Loaded:=FALSE;bAFilm3Loaded:=FALSE;   END_IF


					(*###################### 4th Cone Film Loaded in 2*4  ###################*)


IF bAWrappingCone3OnAuto  AND bAutoModeOn AND b2_4SetHmiSelected AND F_TRIG_3.Q AND NOT  bIWrappingChannelPiston3_End THEN
bAFilm1Loaded_24_4Cone:=TRUE; END_IF

IF bAFilm1Loaded_24_4Cone AND b2_4SetHmiSelected  THEN
bAFilmLoadedCom:=TRUE; bAFilm1Loaded_24_4Cone:=FALSE; END_IF


					(*###################### 5,6th Cone Film Loaded in 2*4   ###################*)


IF bAWrappingCone23OnAuto  AND bAutoModeOn AND b2_4SetHmiSelected AND F_TRIG_2.Q AND NOT  bIWrappingChannelPiston2_End THEN
bAFilm1Loaded_24_5Cone:=TRUE; END_IF
IF bAWrappingCone23OnAuto  AND bAutoModeOn AND b2_4SetHmiSelected  AND F_TRIG_3.Q AND NOT  bIWrappingChannelPiston3_End THEN
bAFilm1Loaded_24_6Cone:=TRUE; END_IF

IF bAFilm1Loaded_24_6Cone AND bAFilm1Loaded_24_5Cone AND b2_4SetHmiSelected THEN
 bAFilmLoadedCom:=TRUE; bAFilm1Loaded_24_6Cone:=FALSE; bAFilm1Loaded_24_5Cone:=FALSE; END_IF


					(*###################### 7,8th Cone Film Loaded in 2*4   ###################*)


IF bAWrappingCone23OnAuto1  AND bAutoModeOn AND b2_4SetHmiSelected AND F_TRIG_2.Q AND NOT  bIWrappingChannelPiston2_End THEN
bAFilm1Loaded_24_7Cone:=TRUE; END_IF
IF bAWrappingCone23OnAuto1  AND bAutoModeOn AND b2_4SetHmiSelected AND F_TRIG_3.Q AND NOT  bIWrappingChannelPiston3_End THEN
bAFilm1Loaded_24_8Cone:=TRUE; END_IF

IF bAFilm1Loaded_24_8Cone AND bAFilm1Loaded_24_7Cone AND b2_4SetHmiSelected  THEN
 bAFilmLoadedCom:=TRUE; bAFilm1Loaded_24_8Cone:=FALSE; bAFilm1Loaded_24_7Cone:=FALSE; END_IF


IF bErrorReset AND bAutoModeOn THEN
 bAFilm1Loaded:=FALSE; bAFilm2Loaded:=FALSE;bAFilm3Loaded:=FALSE;
bAFilm1Loaded_24_8Cone:=FALSE; bAFilm1Loaded_24_7Cone:=FALSE;
bAFilm1Loaded_24_6Cone:=FALSE; bAFilm1Loaded_24_5Cone:=FALSE;
bAFilm1Loaded_24_4Cone:=FALSE; END_IF
END_PROGRAM

(* POU Auto/HMI, ST *)
PROGRAM HMI
VAR

 FB_DateTime_1: FB_DateTime;

	test: WORD;
	Temp1: WORD;
	Temp2: WORD;
	Temp3: WORD;
	Temp4: WORD;
	bAminutes: BOOL;
	bAminutesHmi: WORD;
	bAminutes1stHalf1Hmi: WORD;
	bAminute1stHalf: BOOL;
	bAminutes2ndHalf1Hmi: WORD;
	bAminute2ndHalf: BOOL;
	tes1: INT;
	test2THEN: INT;
	test2: INT;
	bAShift1HourTemp: BOOL;

		wTodayToHmiTemp: STRING;
	TextCol:INT;

	R_TRIG1: R_TRIG;
	NewStep: INT;
	PgmNoDis2: INT;
	MCRunning: BOOL;
	sHour: STRING;
	sTimeTemp1: STRING;
	sMinute: STRING;
	sSecond: STRING;
	sTIMEtemp2: STRING;
	sTIMETemp3: STRING;
	R_TRIG_3: R_TRIG;
	wTodayToHmiFinal: STRING;
END_VAR
(*=========Actual torque to HMI logic===============*)


iTorqueActHmi:= (iTorqueAct );




	sMillNameHmi;
	sAddressLine1Hmi;
	sAddressLine2Hmi;
	sAddressLine3Hmi;
	sCityTownHmi;
	sCountryHmi;


(*==================Logic for  Configuration In Hmi ========================*)

(*=========Empty Cone Enable===============*)

IF bEmptyConeSubOnHmi THEN bEmptyConeSubEnabled:=TRUE; END_IF

IF bEmptyConeSubOffHmi THEN bEmptyConeSubEnabled:=FALSE; END_IF

(*=========Auto Retrival Unit Enable===============*)



IF bAutoRetrivalOnHmi THEN bAutoRetrivalEnabled:=TRUE; END_IF

IF bAutoRetrivalOffHmi THEN bAutoRetrivalEnabled:=FALSE; END_IF


(*=========Printing  Enable===============*)


IF bPrintAutoOnHmi THEN bPrintAutoEnabled:=TRUE; END_IF


IF bPrintAutoOffHmi THEN bPrintAutoEnabled:=FALSE; END_IF

(*=========Print Default weight  Enable===============*)


IF PrintDefaultWeightOnHmi THEN  PrintDefaultWeightOnEnabled:=TRUE; END_IF

IF PrintDefaultWeightOffHmi THEN  PrintDefaultWeightOnEnabled:=FALSE; END_IF

(*=========Negative Tolerance Enable===============*)

IF NegToleranceOnHmi THEN NegToleranceEnabled:=TRUE; END_IF

IF NegToleranceOffHmi THEN NegToleranceEnabled:=FALSE; END_IF

(*======================= RTC==============================*)

FB_DateTime_1(NET_ID:='5.17.63.202.1.1 ' , DATE_TIME=> );

DateTimeVar:=FB_DateTime_1.DATE_TIME;

(*===== Current Date to Hmi and Reports=========*)


wTodayToHmi:=MID(STR:=DateTimeVar, LEN:=10, POS:=1);
wTodayToHmiFinal:=MID(STR:=DateTimeVar, LEN:=20, POS:=1);

sDATEFinal:=  (wTodayToHmiFinal);
(*=======Current TIME to Reports========*)
sTIME:= CONCAT (sTIMETemp3, sSecond) ;
sTIMETemp3:=CONCAT(sTIMEtemp2, ':');

sTIMEtemp2:=CONCAT( sTIMEtemp1 , sMinute);

sTIMEtemp1:=CONCAT(sHour, ':');

sHour:=DWORD_TO_STRING(FB_DateTime_1.FBLTIME.systemTime.wHour);

sMinute:=DWORD_TO_STRING(FB_DateTime_1.FBLTIME.systemTime.wMinute);

sSecond:=DWORD_TO_STRING(FB_DateTime_1.FBLTIME.systemTime.wSecond);

(*wTodayToHmi:=STRING_TO_WORD(wTodayToHmiTemp);  *)

logDay:= WORD_TO_STRING (FB_DateTime_1.FBLTIME.systemTime.wDay);

FB_DateTime_1.FBLTIME.systemTime.wDayOfWeek;

FB_DateTime_1.FBLTIME.systemTime.wHour;

FB_DateTime_1.FBLTIME.systemTime.wMilliseconds;


FB_DateTime_1.FBLTIME.systemTime.wMinute;

LogMonth:= WORD_TO_STRING (FB_DateTime_1.FBLTIME.systemTime.wMonth);



FB_DateTime_1.FBLTIME.systemTime.wSecond;



LogYear:=WORD_TO_STRING (FB_DateTime_1.FBLTIME.systemTime.wYear);


(*===============Shift Calculation============*)





IF FB_DateTime_1.FBLTIME.systemTime.wHour >= Sfiht1From_Hmi AND FB_DateTime_1.FBLTIME.systemTime.wHour<=Sfiht1To_Hmi THEN
bAShift1Hour:=TRUE;

ELSE
bAShift1Hour:=FALSE;

END_IF



IF FB_DateTime_1.FBLTIME.systemTime.wHour>=Sfiht2From_Hmi AND FB_DateTime_1.FBLTIME.systemTime.wHour <= Sfiht2To_Hmi THEN
bAShift2Hour:=TRUE;
ELSE
bAShift2Hour:=FALSE;
END_IF


IF FB_DateTime_1.FBLTIME.systemTime.wHour>=  Sfiht3From_Hmi AND FB_DateTime_1.FBLTIME.systemTime.wHour<=  Sfiht3To_Hmi THEN
bAShift3Hour:=TRUE;
ELSE
bAShift3Hour:=FALSE;
END_IF

IF bAShift1Hour THEN sShitToReport:='Shift1';
ELSIF bAShift2Hour THEN sShitToReport:='Shift2';
ELSIF bAShift3Hour THEN sShitToReport:='Shift3';
END_IF

IF FB_DateTime_1.FBLTIME.systemTime.wMinute >=Shift1MinFrom_HMI AND  FB_DateTime_1.FBLTIME.systemTime.wMinute<=Shift1MinTo_HMI THEN;
END_IF
IF FB_DateTime_1.FBLTIME.systemTime.wMinute >=Shift2MinFrom_HMI AND  FB_DateTime_1.FBLTIME.systemTime.wMinute<=Shift2MinTo_HMI THEN;
END_IF
IF FB_DateTime_1.FBLTIME.systemTime.wMinute >=Shift3MinFrom_HMI AND  FB_DateTime_1.FBLTIME.systemTime.wMinute<=Shift3MinTo_HMI THEN;
END_IF

IF FB_DateTime_1.FBLTIME.systemTime.wMinute > 0 AND  FB_DateTime_1.FBLTIME.systemTime.wMinute<=59 THEN
bAminutes:=TRUE;
ELSE
bAminutes:=FALSE;
END_IF



IF FB_DateTime_1.FBLTIME.systemTime.wMinute > 0  AND  FB_DateTime_1.FBLTIME.systemTime.wMinute<=29 THEN
bAminute1stHalf:=TRUE;
ELSE
bAminute1stHalf:=FALSE;
END_IF



IF FB_DateTime_1.FBLTIME.systemTime.wMinute > 30  AND  FB_DateTime_1.FBLTIME.systemTime.wMinute<=59 THEN
bAminute2ndHalf:=TRUE;
ELSE
bAminute2ndHalf:=FALSE;
END_IF

		IF FB_DateTime_1.FBLTIME.systemTime.wHour =00 AND FB_DateTime_1.FBLTIME.systemTime.wMinute=00 AND FB_DateTime_1.FBLTIME.systemTime.wSecond = 00 THEN
		bADayStart:=TRUE;
		END_IF


		IF FB_DateTime_1.FBLTIME.systemTime.wHour =23 AND FB_DateTime_1.FBLTIME.systemTime.wMinute=59 AND FB_DateTime_1.FBLTIME.systemTime.wSecond = 59 THEN
		bADayComplete:=TRUE;
		END_IF




(*============================== logic for HMI Configuration ==============================*)



(*============== Empty Cone Substract enable Logic======================*)


IF bEmptyConeSubEnableHMI THEN bAEmptyConeSubEnabled:=TRUE; END_IF

IF bEmptyConeSubDisableHMI THEN bAEmptyConeSubEnabled:=FALSE; END_IF

(*==============AutoRetival enable Logic======================*)


IF bAutoRetrivalEnableHMI THEN bAAutoRetrivalEnabled:=TRUE; END_IF

IF bAutoRetrivalDisableHMI THEN bAAutoRetrivalEnabled:=FALSE; END_IF


(*============== Auto Printing enable Logic======================*)

IF bAutoPrintEnableHMI THEN bAAutoPrintEnabled:=TRUE; END_IF

IF bAutoPrintDisableHMI THEN bAAutoPrintEnabled:=FALSE; END_IF


(*==============Default Weight  Print enable Logic======================*)

IF bDefaultWeighPrintEnableHMI THEN bADefaultWeighPrintEnabled:=TRUE; END_IF

IF bDefaultWeighPrintDisableHMI THEN bADefaultWeighPrintEnabled:=FALSE; END_IF

(*==============Negative Tolerance  enable Logic======================*)

IF bNegToletanceEnableHMI THEN bANegToletanceEnabled:=TRUE; END_IF

IF bNegToletanceDisableHMI THEN bANegToletanceEnabled:=FALSE; END_IF




(*==============================Program Setting On HMI=========================*)

(*============================== Packing Type Selection On HMI==================*)


IF bAutoSealingEnableHMI THEN bAAutoSealEnabled:=TRUE; ELSE  bAAutoSealEnabled:=FALSE; END_IF



(*=========================== Pause & Resume Logic =================*)

(*  IF bAutoModeOn AND bPauseHmi THEN bAPauseSeq:=TRUE; END_IF *)

IF bAutoModeOn AND bResumeHmi THEN bAPauseSeq:=FALSE; END_IF


IF bPauseHmi THEN bAPauseSeq:=TRUE; END_IF

(*=========Sealing Complete Delay from Hmi=======*)
SealComDly;

SealComDlyTemp:=REAL_TO_TIME(SealComDly*1000);

(*================Recipe Variable     PACKING TYPE  ==========*)

	IF sSettingArray[i].bAutoSealing THEN bAutoSealOn:=TRUE; bCartonPackingOn:=FALSE; bPallettePackingOn:=FALSE;
	sPackingTypeHmiTemp:= 'AutoSealing';
	ELSIF sSettingArray[i].bCartonPacking THEN bCartonPackingOn:=TRUE; bAutoSealOn:=FALSE; bPallettePackingOn:=FALSE;
	sPackingTypeHmiTemp:= 'Carton Packing';
	ELSIF sSettingArray[i].bPallettePack THEN bPallettePackingOn:=TRUE;  bCartonPackingOn:=FALSE; bAutoSealOn:=FALSE;
	sPackingTypeHmiTemp:= 'Pallette Packing';
	END_IF

	IF bCreateNew THEN
	bAutoSealOn:=FALSE; bCartonPackingOn:=FALSE; bPallettePackingOn:=FALSE;
	END_IF


(*================Recipe Variable     MATERIAL  TYPE  ==========*)

	IF sSettingArray[i].bCone THEN bConeOn:=TRUE; bCheeseOn:=FALSE;
	sMaterialTypeHmiTemp:= 'Cone';
	ELSIF sSettingArray[i].bCheese THEN bConeOn:=FALSE; bCheeseOn:=TRUE;
	sMaterialTypeHmiTemp:= 'Cheese';
	END_IF
(*
R_TRIG1(CLK:=bCreateNew , Q=> );

	IF R_TRIG1.Q THEN
	i:=i+1;
	END_IF
*)


(*================Logic for Model Name Display in Hmi List=============*)



	 PgmNoDis1:=sSettingArray[0].iPgmNo; PgmNameDis1:=sSettingArray[0].iCount;

	 PgmNoDis2:=sSettingArray[1].iPgmNo; PgmNameDis2:=sSettingArray[1].iCount;

	 PgmNoDis3:=sSettingArray[2].iPgmNo; PgmNameDis3:=sSettingArray[2].iCount;

	 PgmNoDis4:=sSettingArray[3].iPgmNo; PgmNameDis4:=sSettingArray[3].iCount;

	 PgmNoDis5:=sSettingArray[4].iPgmNo; PgmNameDis5:=sSettingArray[4].iCount;

	 PgmNoDis6:=sSettingArray[5].iPgmNo; PgmNameDis6:=sSettingArray[5].iCount;



	IF bModel1Hmi THEN i:=0; END_IF

	IF bModel2Hmi THEN i:=1; END_IF

	IF bModel3Hmi THEN i:=2; END_IF

	IF bModel4Hmi THEN i:=3; END_IF

	IF bModel5Hmi THEN i:=4; END_IF

	IF bModel6Hmi THEN i:=5; END_IF


CASE NewStep OF
	0:	IF bCreateNew THEN NewStep:=NewStep+1; END_IF


	1:	IF sSettingArray[0].sDescription=''  THEN
		 i:=0;
		NewStep:=0;
		ELSE
		NewStep:=NewStep+1;
		END_IF

	2:	IF sSettingArray[1].sDescription=''  THEN
		 i:=1;
		NewStep:=0;
		ELSE
		NewStep:=NewStep+1;
		END_IF

	3:	IF sSettingArray[2].sDescription=''  THEN
		 i:=2;
		NewStep:=0;
		ELSE
		NewStep:=NewStep+1;
		END_IF

	4:	IF sSettingArray[3].sDescription=''  THEN
		 i:=3;
		NewStep:=0;
		ELSE
		NewStep:=NewStep+1;
		END_IF


	5:	IF sSettingArray[4].sDescription=''  THEN
		 i:=4;
		NewStep:=0;
		ELSE
		NewStep:=NewStep+1;
		END_IF

	6:	IF sSettingArray[5].sDescription=''  THEN
		 i:=5;
		NewStep:=0;
		ELSE
		NewStep:=NewStep+1;
		END_IF

	7:IF sSettingArray[6].sDescription=''  THEN
		 i:=6;
		NewStep:=0;
		ELSE
		NewStep:=NewStep+1;
		END_IF

	8:	IF sSettingArray[7].sDescription=''  THEN
		 i:=7;
		NewStep:=0;
		ELSE
		NewStep:=NewStep+1;
		END_IF







END_CASE



IF bCreateNew THEN

		Pgm_NoHmi:=0;
		sDescriptionHmi:='';
		iCountHmi:='';
		iLotNoHmi:=0;
		iCartoNoHmi:=0;
		sPackingTypeHmiTemp:='';
		sMaterialTypeHmiTemp:='';
		iConeDiaHmi:=0;
		iHieghtHmi:=0;
		iWeightHmi:=0;
		iTipColorHmi:='';
		iNoOfRowsHmi:=0;
		iNoOfColoumsHmi:=0;
		NoOfLayersHmi:=0;
		iCortonWeightHmi:=0;
		iCartonHmi:=0;
		iLenghtHmi:=0;
		iNoOfConeHmi:=0;
		iNetWeightHmi:=0;
		GrossWeightHmi:=0;
		NetToleranceHmi:=0;
		 rGrossTollHmi:=0;

END_IF








IF bIKeySwitch AND NOT MCRunning THEN bEditRecipeEnabled:=FALSE; ELSE bEditRecipeEnabled:=TRUE; END_IF
(*
IF bRetUnitAStart OR bRetUnitBStart  AND auto
*)
(*============	PLC Variable moving to NOV RAM Variable  ================*)


IF bSaveRecipeHmi THEN


		sSettingArray[i].iPgmNo:=Pgm_NoHmi;
		sSettingArray[i].sDescription:=sDescriptionHmi;
		sSettingArray[i].iCount:=iCountHmi;
		sSettingArray[i].iLotNo:=iLotNoHmi;
		sSettingArray[i].iCartonNo:=iCartoNoHmi;
		sSettingArray[i].iConeDia:=iConeDiaHmi;
		sSettingArray[i].iConeHight:=iHieghtHmi;
		sSettingArray[i].iConeWeight:=iWeightHmi;
		sSettingArray[i].iTipColor:=iTipColorHmi;
		sSettingArray[i].iNoOfRows:=iNoOfRowsHmi;
		sSettingArray[i].iNoOfColoumns:=iNoOfColoumsHmi;
		sSettingArray[i].iNoOfLayers:=NoOfLayersHmi;
		sSettingArray[i].iCartonwidth:=iCortonWeightHmi;
		sSettingArray[i].iCartonHight:=iCartonHmi;
		sSettingArray[i].iCartonLength:=iLenghtHmi;
		sSettingArray[i].iNoOfCones:=iNoOfConeHmi;
		sSettingArray[i].iNetWt:=iNetWeightHmi;
		sSettingArray[i].iGrosswt:=GrossWeightHmi;
		sSettingArray[i].iNetTol:=NetToleranceHmi;
		sSettingArray[i].iGrossTol:= rGrossTollHmi;


END_IF

R_TRIG_3(CLK:= PopUp, Q=> );


IF bloadRecipeHmi  OR R_TRIG_3.Q  THEN
		Pgm_NoHmi:=sSettingArray[i].iPgmNo;
		Var_PgmNo:=Pgm_NoHmi;
		sDescriptionHmi:=sSettingArray[i].sDescription;
		iCountHmi:=sSettingArray[i].iCount;
		Var_Description:= iCountHmi;
		iLotNoHmi:=sSettingArray[i].iLotNo;
		iCartoNoHmi:=sSettingArray[i].iCartonNo;
		sPackingTypeHmiTemp:='';
		sMaterialTypeHmiTemp:='';
		iConeDiaHmi:=sSettingArray[i].iConeDia;
		iHieghtHmi:=sSettingArray[i].iConeHight;
		iWeightHmi:=sSettingArray[i].iConeWeight;
		iTipColorHmi:=sSettingArray[i].iTipColor;
		iNoOfRowsHmi:=sSettingArray[i].iNoOfRows;
		iNoOfColoumsHmi:=sSettingArray[i].iNoOfColoumns;
		NoOfLayersHmi:=sSettingArray[i].iNoOfLayers;
		iCortonWeightHmi:=sSettingArray[i].iCartonwidth;
		iCartonHmi:=sSettingArray[i].iCartonHight;
		iLenghtHmi:=sSettingArray[i].iCartonLength;
		iNoOfConeHmi:=sSettingArray[i].iNoOfCones;
		iNetWeightHmi:=sSettingArray[i].iNetWt;
		GrossWeightHmi:=sSettingArray[i].iGrosswt;
		NetToleranceHmi:=sSettingArray[i].iNetTol;
		 rGrossTollHmi:=sSettingArray[i].iGrossTol;

END_IF
END_PROGRAM

(* POU Auto/RowStopperMotor, ST *)
PROGRAM RowStopperMotor
VAR
	bAModelRest: BOOL;
	step1: INT;
	bQARowStopperMotorFwd1: BOOL;
	R_TRIG1: R_TRIG;
	TON1temp: TON;
	TON1temp1: TON;

	step2: INT;
	TONTemp6: TON;
	TON1temp4: TON;
	TONTemp5: TON;
	test1: BOOL;
	bA2_4RowMoveStarted: BOOL;
	bQARowStopperMotorRev2: BOOL;
	bQARowStopperMotorFwd2: BOOL;
	tRevOffDly: TON;
	tRevOnDly1: TON;
	ColumnStopperInHome: BOOL;
	bA2_3MoveStarted: BOOL;
	bQARowStopperMotorRev3: BOOL;
	bQARowStopperMotorFwd3: BOOL;
	RevOffDly23: TON;
	b23CheckDly: TON;
	tRowStopperHomeDly: TON;
	bQARowStopperMotorRevAuto: BOOL;
	step4: INT;
	bAMove2_4Position: BOOL;
	bAMove2_3Position: BOOL;
	bAProductonStart: BOOL;
	R_TRIG_1: R_TRIG;
	b2_3FirstMoveStart: BOOL;
	TON_1: TON;
	step3: INT;
	bA2_3MoveEnable: BOOL;
	TON_2: TON;
	test: BOOL;
	FwdOffDly23: TON;
	TON_3: TON;
	TON_4: TON;
	TON_5: TON;
	TON1_6: TON;
	R_TRIG_2: R_TRIG;
	b2_4FirstMoveStart: BOOL;
	bA2_4MoveEnable: BOOL;
	RevStartT: TON;
	Step5: INT;
	bARowStopperMotorRevStartTEMP: BOOL;
	bRowStopperRev: BOOL;
	testTemp: BOOL;
	bRowStopperRevtemp: BOOL;
	bAConeOnMatrixConv1: BOOL;
	bAConeOnMatrixConv2: BOOL;
	TON_Mx: TON;
END_VAR
VAR_INPUT
	RowStopperInHome: BOOL;
END_VAR
VAR_OUTPUT
	test2: BOOL;
END_VAR
bQARowStopperMotorForward:= ( bQARowStopperMotorFwd1 OR  bQARowStopperMotorFwd2 OR bQARowStopperMotorFwd3  ) ;
bQARowStopperMotorReverse:= ( bQARowStopperMotorRev1 OR bQARowStopperMotorRev2 OR bQARowStopperMotorRev3 OR bQARowStopperMotorRevAuto OR bRowStopperGoRst ) ;



 IF ((* bAModelRest *)  bRowStopperGoHome OR bRowStopperGoHome1 OR bIntRowStopper )  THEN
bRowStopperRev:=TRUE;
ELSE
bRowStopperRev:=FALSE;
END_IF


CASE step2 OF

	0:	IF bRowStopperRev AND NOT bIRowStopperHome AND   bAutoModeOn   THEN
		bQARowStopperMotorFwd1:=TRUE;
		bRowStopperAt23Pos:=FALSE;
		bRowStopperAt24Pos:=FALSE;
		step2:=step2+1;
		END_IF


	1:	TON1temp4(IN:=TRUE  , PT:=t#1s , Q=> , ET=> );
		IF TON1temp4.Q THEN  step2:=step2+1; END_IF


	2:	bQARowStopperMotorFwd1:=FALSE;
		bAModelRest:=FALSE;
		bRowStopperGoHome:=FALSE;
		bRowStopperGoHome1:=FALSE;
		bIntRowStopper:=FALSE;
		step2:=step2+1;

	3:	RevStartT(IN:=TRUE , PT:=T#1s , Q=> , ET=> );
		IF RevStartT.Q THEN step2:=step2+1; END_IF

	4:	bQARowStopperMotorRev1:=TRUE;
		 step2:=step2+1;

	5:	IF bIRowStopperHome  THEN
		bQARowStopperMotorRev1:=FALSE;
		step2:=0;
		END_IF



END_CASE


IF ( b2_4FirstMoveStart OR bAMove2_4Position OR bGripperUnitOver ) AND  b2_4SetHmiSelected THEN

bA2_4MoveEnable:=TRUE;
ELSE
bA2_4MoveEnable:=FALSE;
END_IF






CASE step1 OF

	0:	IF  bA2_4MoveEnable  AND NOT bIRowStopper3  AND    bIRowStopperHome AND bAutoModeOn AND  NOT bAPauseSeq  THEN
		step1:=step1+1;  END_IF

	1:	step1:=step1+1;


	2:	bA2_4RowMoveStarted:=TRUE;
		bQARowStopperMotorRev2:=FALSE;
		bQARowStopperMotorFwd2:=TRUE;
		bAMove2_4Position:=FALSE;
		TON1_6(IN:=FALSE);
		bGripperUnitOver:=FALSE;step1:=step1+1;

	3:	IF NOT bAPauseSeq THEN step1:=step1+1; END_IF


	4:	 IF bIRowStopper3 THEN
		TON_Mx(IN:=FALSE);
		step1:=step1+1;
		END_IF

	5:	bQARowStopperMotorFwd2:=FALSE; step1:=step1+1;


	6:	IF bIRowStopper3 AND b2_4SetHmiSelected THEN TON_Mx(IN:=TRUE , PT:=T#1s , Q=> , ET=> );
		IF TON_Mx.Q THEN step1:=step1+1;END_IF END_IF


	7:	IF NOT bIRowConeDetection THEN
		b2_4FirstMoveStart:=FALSE;
		bRowStopperAt24Pos:=TRUE;
		bRowStopperIntOver:=TRUE;
		TON_Mx(IN:=FALSE);
		bA2_4RowMoveStarted:=FALSE;
		  step1:=0;
		END_IF


END_CASE







IF ( b2_3FirstMoveStart OR bAMove2_3Position OR(* bRowStopperMoveAftrInt *) bGripperUnitOver )    AND b2_3SetHmiSelected THEN

bA2_3MoveEnable:=TRUE;
ELSE
bA2_3MoveEnable:=FALSE;
END_IF


CASE step3 OF

	0:	IF bA2_3MoveEnable AND NOT bIRowStopper2  AND    bIRowStopperHome  AND NOT bAPauseSeq    THEN
		b23CheckDly(IN:=FALSE);
		TON_5(IN:=FALSE);
		 step3:=step3+1;
		 END_IF

	1:	 step3:=step3+1;

	2:	bA2_3MoveStarted:=TRUE;
		bRowStopperMoveAftrInt:=FALSE;
		bGripperUnitOver:=FALSE;
		bAMove2_3Position:=FALSE;
		bQARowStopperMotorRev3:=FALSE;
		bQARowStopperMotorFwd3:=TRUE;
		step3:=step3+1;

	3:	 step3:=step3+1;

	4:	IF bIRowStopper2 THEN
		TON_Mx(IN:=FALSE);
		step3:=step3+1;
		END_IF

	5:	bQARowStopperMotorFwd3:=FALSE;

		TON_1(IN:=FALSE);
		step3:=step3+1;

	6:	IF bIRowStopper2 THEN TON_Mx(IN:=TRUE , PT:=T#1s , Q=> , ET=> );
		IF TON_Mx.Q THEN step3:=step3+1;END_IF
		END_IF

	7: 	IF NOT bIRowConeDetection THEN
 		bA2_3MoveStarted:=FALSE;
		bRowStopperAt23Pos:=TRUE;
		b2_3FirstMoveStart:=FALSE;
		bRowStopperIntOver:=TRUE;
		TON_Mx(IN:=FALSE);
		step3:=0;END_IF

END_CASE


			(*=====.Cone on Matrix Conveyer======*)

IF (bA2_3MoveStarted OR bA2_4RowMoveStarted) AND (NOT bIRowStopper2 OR NOT bIRowStopper3 ) AND bIRowConeDetection THEN bAConeOnMatrixConv1:=TRUE; END_IF
IF (bA2_3MoveStarted OR bA2_4RowMoveStarted) AND (bIRowStopper2 OR bIRowStopper3 ) AND bIRowConeDetection THEN bAConeOnMatrixConv2:=TRUE; END_IF

IF 	bAConeOnMatrixConv1 OR	bAConeOnMatrixConv2  THEN
	bAConeOnMatrixConv:=TRUE ;sMatrixConvStatus:='Clear Cone At Matrix Conveyor'; bAConeOnMatrixConv1:=FALSE; bAConeOnMatrixConv2:=FALSE;  END_IF

IF bAConeOnMatrixConv AND bAutoModeOn AND bErrorReset AND NOT bIRowConeDetection  THEN
sMatrixConvStatus:='Continue Machine Operation '; bAConeOnMatrixConv:=FALSE;END_IF



(*===================== Auto Logic================*)


CASE step4 OF

	0:	IF( bARowStopperMotorRevStart ) AND bAutoModeOn THEN
		bAMove2_4Position:=FALSE;
		bRowStopperAt23Pos:=FALSE;
		bRowStopperAt24Pos:=FALSE;
		tRowStopperHomeDly(IN:=TRUE , PT:= t#1s , Q=> , ET=> );
		IF tRowStopperHomeDly.Q THEN   step4:=step4+1; END_IF
		END_IF

	1:	step4:=step4+1;


	2:	IF tRowStopperHomeDly.Q AND bAutoModeOn  AND NOT bAPauseSeq   THEN
		bQARowStopperMotorRevAuto:=TRUE;
		bARowStopperMotorRevStart:=FALSE;
		TON_2(IN:=FALSE);
		step4:=step4+1;
		END_IF

	3:	 step4:=step4+1;

	4:	IF bAutoModeOn AND bIRowStopperHome  THEN
		bQARowStopperMotorRevAuto:=FALSE;
		bAServoFwdStart:=TRUE;
		tRowStopperHomeDly(IN:=FALSE);
		step4:=step4+1;
		END_IF

	5:	 step4:=step4+1;

	6:	IF  bIGripperVerticalEnd THEN
		step4:=step4+1;
		END_IF

	7:	IF NOT bIGripperVerticalEnd   AND NOT bAPauseSeq   THEN
		step4:=step4+1;
		END_IF


	8:	 step4:=step4+1;

	9:	TON_2(IN:=TRUE , PT:=T#3S , Q=> , ET=> );
		IF TON_2.Q  THEN bAServoUpDone:=TRUE; step4:=step4+1; END_IF

	10:	 step4:=step4+1;


	11:	IF  bAutoModeOn AND  bAServoUpDone  AND b2_4SetHmiSelected THEN
		step4:=12;
		ELSIF  bAutoModeOn AND  bAServoUpDone AND b2_3SetHmiSelected THEN
		step4:=14;
		END_IF


	12:	 step4:=step4+1;

	13:	 bAMove2_4Position:=TRUE;
		step4:=16;

	14:	 step4:=step4+1;

	15:	bAMove2_3Position:=TRUE;
		step4:=step4+1;

	16:	 step4:=step4+1;

	17:	bAServoUpDone:=FALSE;
		step4:=0;

END_CASE

(*

R_TRIG_1(CLK:=b2_3SetHmiSelected , Q=> );


IF R_TRIG_1.Q AND NOT bIRowStopper2 THEN
b2_3FirstMoveStart:=TRUE;

END_IF

*)

R_TRIG_2(CLK:=b2_4SetHmiSelected , Q=> );


IF R_TRIG_2.Q AND NOT bIRowStopper3 THEN
b2_4FirstMoveStart:=TRUE;

END_IF



(*============= Row Stopper Go to Home Logic While Servo Reset==========================*)


CASE Step5 OF
	0:	IF bRowStopperGoHome THEN bRowStopperGoRst:=TRUE; step5:=1; END_IF

	1:	IF bIRowStopperHome THEN  bRowStopperGoHome:=FALSE; bRowStopperGoRst:=FALSE; Step5:=0; END_IF

END_CASE


IF NOT bIEmergencySwitch OR bStopHmi   OR bServoOff  THEN
TON1temp4(IN:=FALSE);
RevStartT(IN:=FALSE);
bA2_4MoveEnable:=FALSE;
bA2_4RowMoveStarted:=FALSE;
bRowStopperAt24Pos:=FALSE;
bA2_3MoveEnable:=FALSE;
b23CheckDly(IN:=FALSE);
bA2_3MoveStarted:=FALSE;
TON_Mx(IN:=FALSE);
bRowStopperAt23Pos:=FALSE;
bRowStopperIntOver:=FALSE;
bAConeOnMatrixConv1:=FALSE;
bAConeOnMatrixConv2:=FALSE;
bAConeOnMatrixConv:=FALSE;
tRowStopperHomeDly(IN:=FALSE);
TON_2(IN:=FALSE);
bAServoFwdStart:=FALSE;
bAServoUpDone:=FALSE;
bAMove2_4Position:=FALSE;
bAMove2_3Position:=FALSE;

bQARowStopperMotorFwd1:=FALSE;
bQARowStopperMotorFwd2:=FALSE;
bQARowStopperMotorFwd3:=FALSE;
bQARowStopperMotorRev1:=FALSE;
bQARowStopperMotorRev2:=FALSE;
bQARowStopperMotorRev3:=FALSE;
bQARowStopperMotorRevAuto:=FALSE;
bRowStopperGoRst:=FALSE;
step2:=0;
step1:=0;
step3:=0;
step4:=0;

END_IF
END_PROGRAM

